	{attribute 'TcIecLibraryType'}
	{attribute 'external_name' := 'F_VN_GetPerspectiveTransformation_GUID_9BE9794E_D7DA_4639_C989_773406D6F2EE'}
	(* Calculate the perspective transformation between four corresponding point pairs. The points mark the corners of the corresponding rectangles. *)
	FUNCTION F_VN_GetPerspectiveTransformation : HRESULT
	VAR_IN_OUT
		aSrcPoints	:	TcVnArray4_Point2_REAL;	(* Source points *)
		aDestPoints	:	TcVnArray4_Point2_REAL;	(* Destination points *)
		aTransformationMatrix	:	TcVnMatrix3x3_LREAL;	(* Resulting transformation matrix *)
	END_VAR
	VAR_INPUT
		hrPrev	:	HRESULT;	(* HRESULT indicating the result of previous operations (If SUCCEEDED(hrPrev) equals false, no operation is executed.) *)
	END_VAR

END_FUNCTION

// Functions/Geometric and Coordinate Transformations/F_VN_Homography

	{attribute 'TcIecLibraryType'}
	{attribute 'external_name' := 'F_VN_Homography_GUID_E5291A1A_EEBB_4859_F9E7_C15E795ADB21'}
	(* Find the homography (perspective transformation) between two planar point sets using RANSAC algorithm. *)
	FUNCTION F_VN_Homography : HRESULT
	VAR_INPUT
		ipSrcPoints	:	ITcVnContainer;	(* Container with at least 4 source points (ContainerType_Vector_TcVnPoint2_REAL) *)
		ipDestPoints	:	ITcVnContainer;	(* Container with destination points (same number as ipSrcPoints, ContainerType_Vector_TcVnPoint2_REAL) *)
	END_VAR
	VAR_IN_OUT
		aPerspectiveTransform	:	TcVnMatrix3x3_LREAL;	(* Returns the perspective transformation matrix, which transforms the source points to the destination points *)
	END_VAR
	VAR_INPUT
		hrPrev	:	HRESULT;	(* HRESULT indicating the result of previous operations (If SUCCEEDED(hrPrev) equals false, no operation is executed.) *)
	END_VAR

END_FUNCTION

// Functions/Geometric and Coordinate Transformations/F_VN_HomographyExp

	{attribute 'TcIecLibraryType'}
	{attribute 'external_name' := 'F_VN_HomographyExp_GUID_CA9C0CB0_39C3_499B_C695_857A7F2AD576'}
	(* Find the homography (perspective transformation) between two planar point sets. (expert function) *)
	FUNCTION F_VN_HomographyExp : HRESULT
	VAR_INPUT
		ipSrcPoints	:	ITcVnContainer;	(* Container with at least 4 source points (ContainerType_Vector_TcVnPoint2_REAL) *)
		ipDestPoints	:	ITcVnContainer;	(* Container with destination points (same number as ipSrcPoints, ContainerType_Vector_TcVnPoint2_REAL) *)
	END_VAR
	VAR_IN_OUT
		aPerspectiveTransform	:	TcVnMatrix3x3_LREAL;	(* Returns the perspective transformation matrix, which transforms the source points to the destination points *)
	END_VAR
	VAR_INPUT
		eAlgorithm	:	ETcVnEstimationAlgorithm;	(* Estimation algorithm *)
		fReprojThreshold	:	LREAL;	(* Maximum allowed reprojection error to treat a point pair as an inlier (only for RANSAC, RHO) *)
		ipInlierMask	:	REFERENCE TO ITcVnContainer;	(* Returns a mask marking the inliers (optional, set to 0 if not required; ContainerType_Vector_SINT; only for RANSAC, LMEDS) *)
		nMaxIterations	:	UDINT;	(* Maximum number of RANSAC iterations *)
		fConfidence	:	LREAL;	(* Confidence (0..1) *)
		hrPrev	:	HRESULT;	(* HRESULT indicating the result of previous operations (If SUCCEEDED(hrPrev) equals false, no operation is executed.) *)
	END_VAR

END_FUNCTION

// Functions/Geometric and Coordinate Transformations/F_VN_InvertAffineTransformation

	{attribute 'TcIecLibraryType'}
	{attribute 'external_name' := 'F_VN_InvertAffineTransformation_GUID_C334F815_EF33_4023_C9C1_C2FEB1CAF8F9'}
	(* Invert a 2D affine transformation matrix. The inverted transformation compensates the affine transformation on an image if it is used in the F_VN_WarpAffine function. *)
	FUNCTION F_VN_InvertAffineTransformation : HRESULT
	VAR_IN_OUT
		aTransformationMatrix	:	TcVnMatrix2x3_LREAL;	(* Source affine transformation matrix *)
		aInvertedTransformationMatrix	:	TcVnMatrix2x3_LREAL;	(* Resulting inverted affine transformation matrix *)
	END_VAR
	VAR_INPUT
		hrPrev	:	HRESULT;	(* HRESULT indicating the result of previous operations (If SUCCEEDED(hrPrev) equals false, no operation is executed.) *)
	END_VAR

END_FUNCTION

// Functions/Geometric and Coordinate Transformations/F_VN_WarpAffine

	{attribute 'TcIecLibraryType'}
	{attribute 'external_name' := 'F_VN_WarpAffine_GUID_78E1DA68_0848_4442_E97A_23AF60C67DC9'}
	(* Apply an affine transformation to an image. *)
	FUNCTION F_VN_WarpAffine : HRESULT
	VAR_INPUT
		ipSrcImage	:	ITcVnImage;	(* Source image *)
		ipDestImage	:	REFERENCE TO ITcVnImage;	(* Destination image (An appropriate image will be created if required.) *)
	END_VAR
	VAR_IN_OUT
		aTransformationMatrix	:	TcVnMatrix2x3_LREAL;	(* Affine transformation matrix *)
	END_VAR
	VAR_INPUT
		hrPrev	:	HRESULT;	(* HRESULT indicating the result of previous operations (If SUCCEEDED(hrPrev) equals false, no operation is executed.) *)
	END_VAR

END_FUNCTION

// Functions/Geometric and Coordinate Transformations/F_VN_PerspectiveTransformation

	{attribute 'TcIecLibraryType'}
	{attribute 'external_name' := 'F_VN_PerspectiveTransformation_GUID_FEECE007_7BAC_4816_C55F_29631736D6C5'}
	(* Apply a perspective transformation (rotation + translation, e.g. from extrinsic calibration) to 3D point coordinates. *)
	FUNCTION F_VN_PerspectiveTransformation : HRESULT
	VAR_INPUT
		ipSrcPoints	:	ITcVnContainer;	(* Container with 3D source points (TcVnPoint3_REAL or TcVnPoint3_LREAL) *)
		ipDestPoints	:	REFERENCE TO ITcVnContainer;	(* Returns the transformed points (same type as ipSrcPoints) *)
	END_VAR
	VAR_IN_OUT
		aRotationMatrix	:	TcVnMatrix3x3_LREAL;	(* 3x3 rotation matrix *)
		aTranslationVector	:	TcVnVector3_LREAL;	(* Translation vector *)
	END_VAR
	VAR_INPUT
		hrPrev	:	HRESULT;	(* HRESULT indicating the result of previous operations (If SUCCEEDED(hrPrev) equals false, no operation is executed.) *)
	END_VAR

END_FUNCTION

// Functions/Geometric and Coordinate Transformations/F_VN_PyramidDown

	{attribute 'TcIecLibraryType'}
	{attribute 'external_name' := 'F_VN_PyramidDown_GUID_FB8B02E5_B7F2_4AD9_D83B_083942D35F0A'}
	(* Downsamples an image to half width and height. *)
	FUNCTION F_VN_PyramidDown : HRESULT
	VAR_INPUT
		ipSrcImage	:	ITcVnImage;	(* Source image *)
		ipDestImage	:	REFERENCE TO ITcVnImage;	(* Destination image (An appropriate destination image will be created if required.) *)
		hrPrev	:	HRESULT;	(* HRESULT indicating the result of previous operations (If SUCCEEDED(hrPrev) equals false, no operation is executed.) *)
	END_VAR

END_FUNCTION

// Functions/Geometric and Coordinate Transformations/F_VN_PyramidUp

	{attribute 'TcIecLibraryType'}
	{attribute 'external_name' := 'F_VN_PyramidUp_GUID_9885070C_2F9E_4CBD_C0E2_B8BDF3FAFC70'}
	(* Upsamples an image to double width and height. *)
	FUNCTION F_VN_PyramidUp : HRESULT
	VAR_INPUT
		ipSrcImage	:	ITcVnImage;	(* Source image *)
		ipDestImage	:	REFERENCE TO ITcVnImage;	(* Destination image (An appropriate destination image will be created if required.) *)
		hrPrev	:	HRESULT;	(* HRESULT indicating the result of previous operations (If SUCCEEDED(hrPrev) equals false, no operation is executed.) *)
	END_VAR

END_FUNCTION

// Functions/Geometric and Coordinate Transformations/F_VN_RemapImageToLogPolarSpace

	{attribute 'TcIecLibraryType'}
	{attribute 'external_name' := 'F_VN_RemapImageToLogPolarSpace_GUID_6E99848D_0ACF_4D69_F527_2E3106AFEFD3'}
	(* Remap an image to log-polar space. *)
	FUNCTION F_VN_RemapImageToLogPolarSpace : HRESULT
	VAR_INPUT
		ipSrcImage	:	ITcVnImage;	(* Source image *)
		ipDestImage	:	REFERENCE TO ITcVnImage;	(* Destination image (Must not be the same as ipSrcImage! An appropriate destination image will be created if required.) *)
	END_VAR
	VAR_IN_OUT
		aCenter	:	TcVnPoint2_REAL;	(* Center point for the transformation *)
	END_VAR
	VAR_INPUT
		hrPrev	:	HRESULT;	(* HRESULT indicating the result of previous operations (If SUCCEEDED(hrPrev) equals false, no operation is executed.) *)
	END_VAR

END_FUNCTION

// Functions/Geometric and Coordinate Transformations/F_VN_RemapImageToLogPolarSpaceExp

	{attribute 'TcIecLibraryType'}
	{attribute 'external_name' := 'F_VN_RemapImageToLogPolarSpaceExp_GUID_9BB5F0DA_4683_4F22_C3F2_6DF6CC34EE46'}
	(* Remap an image to log-polar space. (expert function) *)
	FUNCTION F_VN_RemapImageToLogPolarSpaceExp : HRESULT
	VAR_INPUT
		ipSrcImage	:	ITcVnImage;	(* Source image *)
		ipDestImage	:	REFERENCE TO ITcVnImage;	(* Destination image (Must not be the same as ipSrcImage! An appropriate destination image will be created if required.) *)
	END_VAR
	VAR_IN_OUT
		aCenter	:	TcVnPoint2_REAL;	(* Center point for the transformation *)
	END_VAR
	VAR_INPUT
		fScale	:	LREAL;	(* Magnitude scale parameter, i.e. image width / ln(radius) (set to 0 for auto select) *)
		eInterpolationType	:	ETcVnInterpolationType;	(* Interpolation type *)
		hrPrev	:	HRESULT;	(* HRESULT indicating the result of previous operations (If SUCCEEDED(hrPrev) equals false, no operation is executed.) *)
	END_VAR

END_FUNCTION

// Functions/Geometric and Coordinate Transformations/F_VN_RemapImageToLogPolarSpaceExp2

	{attribute 'TcIecLibraryType'}
	{attribute 'external_name' := 'F_VN_RemapImageToLogPolarSpaceExp2_GUID_D347BCEC_E69F_4A83_E12E_F22818680819'}
	(* Remap an image to log-polar space. (expert function) *)
	FUNCTION F_VN_RemapImageToLogPolarSpaceExp2 : HRESULT
	VAR_INPUT
		ipSrcImage	:	ITcVnImage;	(* Source image *)
		ipDestImage	:	REFERENCE TO ITcVnImage;	(* Destination image (Must not be the same as ipSrcImage! An appropriate destination image will be created if required.) *)
	END_VAR
	VAR_IN_OUT
		aCenter	:	TcVnPoint2_REAL;	(* Center point for the transformation *)
	END_VAR
	VAR_INPUT
		fScale	:	LREAL;	(* Magnitude scale parameter, i.e. image width / ln(radius) (set to 0 for auto select) *)
		eInterpolationType	:	ETcVnInterpolationType;	(* Interpolation type *)
		nDestWidth	:	DINT;	(* Destination image width (set to -1 for source image width, 0 to auto scale to transformed radius, > 0 for a user defined width) *)
		nDestHeight	:	DINT;	(* destination image height (set to -1 for source image height, 0 to auto scale to transformed radius * PI, > 0 for a user defined height) *)
		hrPrev	:	HRESULT;	(* HRESULT indicating the result of previous operations (If SUCCEEDED(hrPrev) equals false, no operation is executed.) *)
	END_VAR

END_FUNCTION

// Functions/Geometric and Coordinate Transformations/F_VN_RemapImageToPolarSpace

	{attribute 'TcIecLibraryType'}
	{attribute 'external_name' := 'F_VN_RemapImageToPolarSpace_GUID_DE45FD10_0322_4630_F43A_30A819E434CD'}
	(* Remap an image to polar space. *)
	FUNCTION F_VN_RemapImageToPolarSpace : HRESULT
	VAR_INPUT
		ipSrcImage	:	ITcVnImage;	(* Source image *)
		ipDestImage	:	REFERENCE TO ITcVnImage;	(* Destination image (Must not be the same as ipSrcImage! An appropriate destination image will be created if required.) *)
	END_VAR
	VAR_IN_OUT
		aCenter	:	TcVnPoint2_REAL;	(* Center point for the transformation *)
	END_VAR
	VAR_INPUT
		hrPrev	:	HRESULT;	(* HRESULT indicating the result of previous operations (If SUCCEEDED(hrPrev) equals false, no operation is executed.) *)
	END_VAR

END_FUNCTION

// Functions/Geometric and Coordinate Transformations/F_VN_RemapImageToPolarSpaceExp

	{attribute 'TcIecLibraryType'}
	{attribute 'external_name' := 'F_VN_RemapImageToPolarSpaceExp_GUID_9860E05D_5A15_4F04_E9E1_22F5EF3B73E2'}
	(* Remap an image to polar space. (expert function) *)
	FUNCTION F_VN_RemapImageToPolarSpaceExp : HRESULT
	VAR_INPUT
		ipSrcImage	:	ITcVnImage;	(* Source image *)
		ipDestImage	:	REFERENCE TO ITcVnImage;	(* Destination image (Must not be the same as ipSrcImage! An appropriate destination image will be created if required.) *)
	END_VAR
	VAR_IN_OUT
		aCenter	:	TcVnPoint2_REAL;	(* Center point for the transformation *)
	END_VAR
	VAR_INPUT
		fMaxRadius	:	LREAL;	(* Maximum radius for the transformation (set to 0 for auto select) *)
		eInterpolationType	:	ETcVnInterpolationType;	(* Interpolation type *)
		hrPrev	:	HRESULT;	(* HRESULT indicating the result of previous operations (If SUCCEEDED(hrPrev) equals false, no operation is executed.) *)
	END_VAR

END_FUNCTION

// Functions/Geometric and Coordinate Transformations/F_VN_RemapImageToPolarSpaceExp2

	{attribute 'TcIecLibraryType'}
	{attribute 'external_name' := 'F_VN_RemapImageToPolarSpaceExp2_GUID_630BAAF6_2143_4E62_F9BA_CD5AAB59C67E'}
	(* Remap an image to polar space. (expert function) *)
	FUNCTION F_VN_RemapImageToPolarSpaceExp2 : HRESULT
	VAR_INPUT
		ipSrcImage	:	ITcVnImage;	(* Source image *)
		ipDestImage	:	REFERENCE TO ITcVnImage;	(* Destination image (Must not be the same as ipSrcImage! An appropriate destination image will be created if required.) *)
	END_VAR
	VAR_IN_OUT
		aCenter	:	TcVnPoint2_REAL;	(* Center point for the transformation *)
	END_VAR
	VAR_INPUT
		fMaxRadius	:	LREAL;	(* Maximum radius for the transformation (set to 0 for auto select) *)
		eInterpolationType	:	ETcVnInterpolationType;	(* Interpolation type *)
		nDestWidth	:	DINT;	(* Destination image width (set to -1 for source image width, 0 to auto scale to transformed radius, > 0 for a user defined width) *)
		nDestHeight	:	DINT;	(* destination image height (set to -1 for source image height, 0 to auto scale to transformed radius * PI, > 0 for a user defined height) *)
		hrPrev	:	HRESULT;	(* HRESULT indicating the result of previous operations (If SUCCEEDED(hrPrev) equals false, no operation is executed.) *)
	END_VAR

END_FUNCTION

// Functions/Geometric and Coordinate Transformations/F_VN_ResizeImage

	{attribute 'TcIecLibraryType'}
	{attribute 'external_name' := 'F_VN_ResizeImage_GUID_ED70CE00_559D_43CE_CB1F_72B9FB8B052F'}
	(* Resize an image using a specific interpolation type. *)
	FUNCTION F_VN_ResizeImage : HRESULT
	VAR_INPUT
		ipSrcImage	:	ITcVnImage;	(* Source image *)
		ipDestImage	:	REFERENCE TO ITcVnImage;	(* Destination image (An appropriate image will be created if required.) *)
		nWidth	:	UDINT;	(* New width *)
		nHeight	:	UDINT;	(* New height *)
		eInterpolationType	:	ETcVnInterpolationType;	(* Interpolation type *)
		hrPrev	:	HRESULT;	(* HRESULT indicating the result of previous operations (If SUCCEEDED(hrPrev) equals false, no operation is executed.) *)
	END_VAR

END_FUNCTION

// Functions/Geometric and Coordinate Transformations/F_VN_ResizeImageExp

	{attribute 'TcIecLibraryType'}
	{attribute 'external_name' := 'F_VN_ResizeImageExp_GUID_377703E0_DC16_4250_DD46_18CED214792B'}
	(* Resize an image using a specific interpolation type while maintaining its aspect ratio. (expert function) *)
	FUNCTION F_VN_ResizeImageExp : HRESULT
	VAR_INPUT
		ipSrcImage	:	ITcVnImage;	(* Source image *)
		ipDestImage	:	REFERENCE TO ITcVnImage;	(* Destination image (An appropriate image will be created if required.) *)
		nWidth	:	UDINT;	(* New width *)
		nHeight	:	UDINT;	(* New height *)
		eInterpolationType	:	ETcVnInterpolationType;	(* Interpolation type *)
		ePaddingMode	:	ETcVnPaddingMode;	(* Image padding mode *)
	END_VAR
	VAR_IN_OUT
		aBorderValue	:	TcVnVector4_LREAL;	(* Border value, if TCVN_PM_LETTERBOX is used *)
	END_VAR
	VAR_INPUT
		hrPrev	:	HRESULT;	(* HRESULT indicating the result of previous operations (If SUCCEEDED(hrPrev) equals false, no operation is executed.) *)
	END_VAR

END_FUNCTION

// Functions/Geometric and Coordinate Transformations/F_VN_RotateImage

	{attribute 'TcIecLibraryType'}
	{attribute 'external_name' := 'F_VN_RotateImage_GUID_8CAB3FB7_5E87_43EF_E423_2C00B8AA20D2'}
	(* Rotate an image by 90, 180, or 270 degrees in clockwise direction. *)
	FUNCTION F_VN_RotateImage : HRESULT
	VAR_INPUT
		ipSrcImage	:	ITcVnImage;	(* Source image *)
		ipDestImage	:	REFERENCE TO ITcVnImage;	(* Destination image (An appropriate image will be created if required.) *)
		eAngle	:	ETcVnRotationAngle;	(* Rotation angle *)
		hrPrev	:	HRESULT;	(* HRESULT indicating the result of previous operations (If SUCCEEDED(hrPrev) equals false, no operation is executed.) *)
	END_VAR

END_FUNCTION

// Functions/Geometric and Coordinate Transformations/F_VN_RotateImageExp

	{attribute 'TcIecLibraryType'}
	{attribute 'external_name' := 'F_VN_RotateImageExp_GUID_A2207F24_DE10_44CD_DD61_03B9D4F8B389'}
	(* Rotate an image by an individual rotation angle in degrees. *)
	FUNCTION F_VN_RotateImageExp : HRESULT
	VAR_INPUT
		ipSrcImage	:	ITcVnImage;	(* Source image *)
		ipDestImage	:	REFERENCE TO ITcVnImage;	(* Destination image (An appropriate image will be created if required.) *)
		fAngleDeg	:	LREAL;	(* Rotation angle in degree (positive: counter-clockwise, negative: clockwise) *)
		bAdjustDestSize	:	BOOL;	(* If true, ipDestImage size is adjusted so that the whole rotated ipSrcImage is contained. Otherwise, ipDestImage size is set to ipSrcImage size. *)
		hrPrev	:	HRESULT;	(* HRESULT indicating the result of previous operations (If SUCCEEDED(hrPrev) equals false, no operation is executed.) *)
	END_VAR

END_FUNCTION

// Functions/Geometric and Coordinate Transformations/F_VN_RotateImageExp2

	{attribute 'TcIecLibraryType'}
	{attribute 'external_name' := 'F_VN_RotateImageExp2_GUID_85F7CE2B_7D57_4E8E_D6F0_120EAB5D6A53'}
	(* Rotate an image by an individual rotation angle in degrees. (expert function) *)
	FUNCTION F_VN_RotateImageExp2 : HRESULT
	VAR_INPUT
		ipSrcImage	:	ITcVnImage;	(* Source image *)
		ipDestImage	:	REFERENCE TO ITcVnImage;	(* Destination image (An appropriate image will be created if required.) *)
		fAngleDeg	:	LREAL;	(* Rotation angle in degree (positive: counter-clockwise, negative: clockwise) *)
		bAdjustDestSize	:	BOOL;	(* If true, ipDestImage size is adjusted so that the whole rotated ipSrcImage is contained. Otherwise, ipDestImage size is set to ipSrcImage size. *)
		eInterpolationType	:	ETcVnInterpolationType;	(* Interpolation method *)
		eBorderInterpolation	:	ETcVnBorderInterpolationMethod;	(* Border interpolation method (ISOLATED not supported) *)
	END_VAR
	VAR_IN_OUT
		aBorderValue	:	TcVnVector4_LREAL;	(* Border value, if CONSTANT is used *)
	END_VAR
	VAR_INPUT
		hrPrev	:	HRESULT;	(* HRESULT indicating the result of previous operations (If SUCCEEDED(hrPrev) equals false, no operation is executed.) *)
	END_VAR

END_FUNCTION

// Functions/Geometric and Coordinate Transformations/F_VN_WarpAffineExp

	{attribute 'TcIecLibraryType'}
	{attribute 'external_name' := 'F_VN_WarpAffineExp_GUID_E5CBC38D_CE6D_4892_FDDC_E6736DBE061C'}
	(* Apply an affine transformation to an image. (expert function) *)
	FUNCTION F_VN_WarpAffineExp : HRESULT
	VAR_INPUT
		ipSrcImage	:	ITcVnImage;	(* Source image *)
		ipDestImage	:	REFERENCE TO ITcVnImage;	(* Destination image (An appropriate image will be created if required.) *)
	END_VAR
	VAR_IN_OUT
		aTransformationMatrix	:	TcVnMatrix2x3_LREAL;	(* Affine transformation matrix *)
	END_VAR
	VAR_INPUT
		nDestWidth	:	UDINT;	(* Width of the destination image *)
		nDestHeight	:	UDINT;	(* Height of the destination image *)
		eInterpolationType	:	ETcVnInterpolationType;	(* Interpolation method *)
		bWarpInverse	:	BOOL;	(* Handle aTransformationMatrix as the inverse transformation *)
		eBorderInterpolation	:	ETcVnBorderInterpolationMethod;	(* Border interpolation method (ISOLATED not supported) *)
		fBorderValue	:	LREAL;	(* Border value, if CONSTANT is used *)
		hrPrev	:	HRESULT;	(* HRESULT indicating the result of previous operations (If SUCCEEDED(hrPrev) equals false, no operation is executed.) *)
	END_VAR

END_FUNCTION

// Functions/Geometric and Coordinate Transformations/F_VN_WarpAffine_Container

	{attribute 'TcIecLibraryType'}
	{attribute 'external_name' := 'F_VN_WarpAffine_Container_GUID_BDA2D4B3_B51A_4A2F_C820_697FB0178013'}
	(* Apply an affine transformation to a container of 2D points. *)
	FUNCTION F_VN_WarpAffine_Container : HRESULT
	VAR_INPUT
		ipSrcPoints	:	ITcVnContainer;	(* Source points (ContainerType_Vector_TcVnPoint2_DINT or ContainerType_Vector_TcVnPoint2_REAL or ContainerType_Vector_TcVnPoint2_LREAL) *)
		ipDestPoints	:	REFERENCE TO ITcVnContainer;	(* Returns the transformed points (same type ID as ipSrcPoints; Non-zero interface pointers are reused.) *)
	END_VAR
	VAR_IN_OUT
		aTransformationMatrix	:	TcVnMatrix2x3_LREAL;	(* Affine transformation matrix *)
	END_VAR
	VAR_INPUT
		hrPrev	:	HRESULT;	(* HRESULT indicating the result of previous operations (If SUCCEEDED(hrPrev) equals false, no operation is executed.) *)
	END_VAR

END_FUNCTION

// Functions/Geometric and Coordinate Transformations/F_VN_WarpAffine_Point

	{attribute 'TcIecLibraryType'}
	{attribute 'external_name' := 'F_VN_WarpAffine_Point_GUID_0C65AB93_8901_4F57_F455_A874377D5041'}
	(* Apply an affine transformation to a 2D point. *)
	FUNCTION F_VN_WarpAffine_Point : HRESULT
	VAR_IN_OUT
		aSrcPoint	:	TcVnPoint2_LREAL;	(* Source point *)
		aDestPoint	:	TcVnPoint2_LREAL;	(* Destination point *)
		aTransformationMatrix	:	TcVnMatrix2x3_LREAL;	(* Affine transformation matrix *)
	END_VAR
	VAR_INPUT
		hrPrev	:	HRESULT;	(* HRESULT indicating the result of previous operations (If SUCCEEDED(hrPrev) equals false, no operation is executed.) *)
	END_VAR

END_FUNCTION

// Functions/Geometric and Coordinate Transformations/F_VN_WarpAffine_Rectangle

	{attribute 'TcIecLibraryType'}
	{attribute 'external_name' := 'F_VN_WarpAffine_Rectangle_GUID_5C0D29CF_C44A_4C24_F34A_859F4FD8ADB8'}
	(* Use an affine transform to warp a rectangle. *)
	FUNCTION F_VN_WarpAffine_Rectangle : HRESULT
	VAR_INPUT
		nTopLeftX	:	UDINT;	(* x coordinate of the top left corner *)
		nTopLeftY	:	UDINT;	(* y coordinate of the top left corner *)
		nBottomRightX	:	UDINT;	(* x coordinate of the bottom right corner *)
		nBottomRightY	:	UDINT;	(* y coordinate of the bottom right corner *)
		ipDestPoints	:	REFERENCE TO ITcVnContainer;	(* Returns the 4 transformed points (ContainerType_Vector_TcVnPoint2_REAL) *)
	END_VAR
	VAR_IN_OUT
		aTransformationMatrix	:	TcVnMatrix2x3_LREAL;	(* Affine transformation matrix *)
	END_VAR
	VAR_INPUT
		hrPrev	:	HRESULT;	(* HRESULT indicating the result of previous operations (If SUCCEEDED(hrPrev) equals false, no operation is executed.) *)
	END_VAR

END_FUNCTION

// Functions/Geometric and Coordinate Transformations/F_VN_WarpPerspective

	{attribute 'TcIecLibraryType'}
	{attribute 'external_name' := 'F_VN_WarpPerspective_GUID_FA579732_BEC2_4958_E42E_5F92911D7AE0'}
	(* Apply a perspective transformation to an image. *)
	FUNCTION F_VN_WarpPerspective : HRESULT
	VAR_INPUT
		ipSrcImage	:	ITcVnImage;	(* Source image *)
		ipDestImage	:	REFERENCE TO ITcVnImage;	(* Destination image (An appropriate image will be created if required.) *)
	END_VAR
	VAR_IN_OUT
		aTransformationMatrix	:	TcVnMatrix3x3_LREAL;	(* Perspective transformation matrix *)
	END_VAR
	VAR_INPUT
		hrPrev	:	HRESULT;	(* HRESULT indicating the result of previous operations (If SUCCEEDED(hrPrev) equals false, no operation is executed.) *)
	END_VAR

END_FUNCTION

// Functions/Geometric and Coordinate Transformations/F_VN_WarpPerspective_Container

	{attribute 'TcIecLibraryType'}
	{attribute 'external_name' := 'F_VN_WarpPerspective_Container_GUID_F182FCB6_9954_46A8_C212_0E4575B35202'}
	(* Apply a perspective transformation to a container of 2D points. *)
	FUNCTION F_VN_WarpPerspective_Container : HRESULT
	VAR_INPUT
		ipSrcPoints	:	ITcVnContainer;	(* Source points (ContainerType_Vector_TcVnPoint2_DINT or ContainerType_Vector_TcVnPoint2_REAL or ContainerType_Vector_TcVnPoint2_LREAL) *)
		ipDestPoints	:	REFERENCE TO ITcVnContainer;	(* Returns the transformed points (same type ID as ipSrcPoints; Non-zero interface pointers are reused.) *)
	END_VAR
	VAR_IN_OUT
		aTransformationMatrix	:	TcVnMatrix3x3_LREAL;	(* Perspective transformation matrix *)
	END_VAR
	VAR_INPUT
		hrPrev	:	HRESULT;	(* HRESULT indicating the result of previous operations (If SUCCEEDED(hrPrev) equals false, no operation is executed.) *)
	END_VAR

END_FUNCTION

// Functions/Geometric and Coordinate Transformations/F_VN_WarpPerspectiveExp

	{attribute 'TcIecLibraryType'}
	{attribute 'external_name' := 'F_VN_WarpPerspectiveExp_GUID_0101B598_6EE4_4C4D_F167_907DFB52670E'}
	(* Apply a perspective transformation to an image. (expert function) *)
	FUNCTION F_VN_WarpPerspectiveExp : HRESULT
	VAR_INPUT
		ipSrcImage	:	ITcVnImage;	(* Source image *)
		ipDestImage	:	REFERENCE TO ITcVnImage;	(* Destination image (An appropriate image will be created if required.) *)
	END_VAR
	VAR_IN_OUT
		aTransformationMatrix	:	TcVnMatrix3x3_LREAL;	(* Perspective transformation matrix *)
	END_VAR
	VAR_INPUT
		nDestWidth	:	UDINT;	(* Width of the destination image *)
		nDestHeight	:	UDINT;	(* Height of the destination image *)
		eInterpolationType	:	ETcVnInterpolationType;	(* Interpolation method *)
		bWarpInverse	:	BOOL;	(* Handle aTransformationMatrix as the inverse transformation *)
		eBorderInterpolation	:	ETcVnBorderInterpolationMethod;	(* Border interpolation method (ISOLATED not supported) *)
		fBorderValue	:	LREAL;	(* Border value, if CONSTANT is used *)
		hrPrev	:	HRESULT;	(* HRESULT indicating the result of previous operations (If SUCCEEDED(hrPrev) equals false, no operation is executed.) *)
	END_VAR

END_FUNCTION

// Functions/Geometric and Coordinate Transformations/F_VN_WarpPerspective_Point

	{attribute 'TcIecLibraryType'}
	{attribute 'external_name' := 'F_VN_WarpPerspective_Point_GUID_0ADF8ADE_46B9_4EEE_EE54_6AF0F99DCBC8'}
	(* Apply a perspective transformation to a 2D point. *)
	FUNCTION F_VN_WarpPerspective_Point : HRESULT
	VAR_IN_OUT
		aSrcPoint	:	TcVnPoint2_LREAL;	(* Source point *)
		aDestPoint	:	TcVnPoint2_LREAL;	(* Destination point *)
		aTransformationMatrix	:	TcVnMatrix3x3_LREAL;	(* Perspective transformation matrix *)
	END_VAR
	VAR_INPUT
		hrPrev	:	HRESULT;	(* HRESULT indicating the result of previous operations (If SUCCEEDED(hrPrev) equals false, no operation is executed.) *)
	END_VAR

END_FUNCTION

// Functions/Geometric and Coordinate Transformations/F_VN_WarpPerspective_Rectangle

	{attribute 'TcIecLibraryType'}
	{attribute 'external_name' := 'F_VN_WarpPerspective_Rectangle_GUID_FCB2B455_A681_4AD4_F5F7_27725716AA61'}
	(* Use a perspective transform to warp a rectangle. *)
	FUNCTION F_VN_WarpPerspective_Rectangle : HRESULT
	VAR_INPUT
		nTopLeftX	:	UDINT;	(* x coordinate of the top left corner *)
		nTopLeftY	:	UDINT;	(* y coordinate of the top left corner *)
		nBottomRightX	:	UDINT;	(* x coordinate of the bottom right corner *)
		nBottomRightY	:	UDINT;	(* y coordinate of the bottom right corner *)
		ipDestPoints	:	REFERENCE TO ITcVnContainer;	(* Returns the 4 transformed points (ContainerType_Vector_TcVnPoint2_REAL) *)
	END_VAR
	VAR_IN_OUT
		aTransformationMatrix	:	TcVnMatrix3x3_LREAL;	(* Perspective transformation matrix *)
	END_VAR
	VAR_INPUT
		hrPrev	:	HRESULT;	(* HRESULT indicating the result of previous operations (If SUCCEEDED(hrPrev) equals false, no operation is executed.) *)
	END_VAR

END_FUNCTION

// Functions/Image Color and Contrast Processing/F_VN_ApplyColorMap

	{attribute 'TcIecLibraryType'}
	{attribute 'external_name' := 'F_VN_ApplyColorMap_GUID_6A737126_4D72_4BCB_EC05_C06460642509'}
	(* Apply a color map to a gray-level image. *)
	FUNCTION F_VN_ApplyColorMap : HRESULT
	VAR_INPUT
		ipSrcImage	:	ITcVnImage;	(* Source image (TCVN_ET_USINT or TCVN_ET_UINT, 1 channel) *)
		ipDestImage	:	REFERENCE TO ITcVnImage;	(* Returns the colored image (TCVN_ET_USINT, 3 channel. An appropriate image will be created if required.) *)
		ipColorMap	:	ITcVnContainer;	(* Color map to be applied to ipSrcImage (ContainerType_Vector_TcVnVector3_REAL with 256 or 65536 elements, dependent on ipSrcImage type). Can be either custom or created with F_VN_GenerateColorMap. *)
		hrPrev	:	HRESULT;	(* HRESULT indicating the result of previous operations (If SUCCEEDED(hrPrev) equals false, no operation is executed.) *)
	END_VAR

END_FUNCTION

// Functions/Image Color and Contrast Processing/F_VN_GenerateColorMap

	{attribute 'TcIecLibraryType'}
	{attribute 'external_name' := 'F_VN_GenerateColorMap_GUID_74A0CE66_74B2_42A4_C756_B0F27E943F8E'}
	(* Generates a pre-defined color map. *)
	FUNCTION F_VN_GenerateColorMap : HRESULT
	VAR_INPUT
		ipColorMap	:	REFERENCE TO ITcVnContainer;	(* Returns the color map (ContainerType_Vector_TcVnVector3_REAL with 256 or 65536 elements) *)
		eColorMap	:	ETcVnColorMap;	(* Selects a color map (similar to GNU Octave/MATLAB types) *)
		eColorMapSize	:	ETcVnColorMapSize;	(* Defines how many elements the generated color map should have *)
		hrPrev	:	HRESULT;	(* HRESULT indicating the result of previous operations (If SUCCEEDED(hrPrev) equals false, no operation is executed.) *)
	END_VAR

END_FUNCTION

// Functions/Image Color and Contrast Processing/F_VN_ApplyLut

	{attribute 'TcIecLibraryType'}
	{attribute 'external_name' := 'F_VN_ApplyLut_GUID_68C1FC50_DE6A_4FE0_E3D5_AD24FA9B5417'}
	(* Apply a lookup table to an image to manipulate its colors. *)
	FUNCTION F_VN_ApplyLut : HRESULT
	VAR_INPUT
		ipSrcImage	:	ITcVnImage;	(* Source image (1-4 channels of 8 or 16 bit types SINT, USINT, INT, UINT) *)
		ipDestImage	:	REFERENCE TO ITcVnImage;	(* Returns the result image (same size, type and channels as ipSrcImage. An appropriate image will be created if required.) *)
		ipLut	:	ITcVnContainer;	(* Lookup table with elements matching ipSrcImage type and either 256 (8 bit images) or 65536 (16 bit images) elements. E.g. ContainerType_Vector_USINT for 1-4 channel USINT image (in this case, the same lookup values are used for each channel) or ContainerType_Vector_TcVnVector3_USINT for a 3 channel USINT image (in this case, each channel uses an individual lookup value).
						 *)
		hrPrev	:	HRESULT;	(* HRESULT indicating the result of previous operations (If SUCCEEDED(hrPrev) equals false, no operation is executed.) *)
	END_VAR

END_FUNCTION

// Functions/Image Color and Contrast Processing/F_VN_Clahe

	{attribute 'TcIecLibraryType'}
	{attribute 'external_name' := 'F_VN_Clahe_GUID_5A201C60_0417_4646_D4DD_B850B6060DD9'}
	(* Apply Constrast Limited Adaptive Histogram Equalization. This applies local histogram equalization to individual tiles. *)
	FUNCTION F_VN_Clahe : HRESULT
	VAR_INPUT
		ipSrcImage	:	ITcVnImage;	(* Source image (TCVN_ET_USINT or TCVN_ET_UINT, 1 channel) *)
		ipDestImage	:	REFERENCE TO ITcVnImage;	(* Returns the resulting image (An appropriate image will be created if required.) *)
		hrPrev	:	HRESULT;	(* HRESULT indicating the result of previous operations (If SUCCEEDED(hrPrev) equals false, no operation is executed.) *)
	END_VAR

END_FUNCTION

// Functions/Image Color and Contrast Processing/F_VN_ClaheExp

	{attribute 'TcIecLibraryType'}
	{attribute 'external_name' := 'F_VN_ClaheExp_GUID_E01C29C2_6F3D_4620_E8A1_F87756DA5EF7'}
	(* Apply Constrast Limited Adaptive Histogram Equalization. This applies local histogram equalization to individual tiles. (expert function) *)
	FUNCTION F_VN_ClaheExp : HRESULT
	VAR_INPUT
		ipSrcImage	:	ITcVnImage;	(* Source image (TCVN_ET_USINT or TCVN_ET_UINT, 1 channel) *)
		ipDestImage	:	REFERENCE TO ITcVnImage;	(* Returns the resulting image (An appropriate image will be created if required.) *)
		fClipLimit	:	LREAL;	(* Threshold for contrast limit (set to <= 0 to disable clipping) *)
		nTilesX	:	UDINT;	(* Number of tiles in x direction *)
		nTilesY	:	UDINT;	(* Number of tiles in y direction *)
		hrPrev	:	HRESULT;	(* HRESULT indicating the result of previous operations (If SUCCEEDED(hrPrev) equals false, no operation is executed.) *)
	END_VAR

END_FUNCTION

// Functions/Image Color and Contrast Processing/F_VN_ConvertColorSpace

	{attribute 'TcIecLibraryType'}
	{attribute 'external_name' := 'F_VN_ConvertColorSpace_GUID_0C9A6943_44C8_4F3F_E050_0540D257B30D'}
	(* Convert image from one color space to another. *)
	FUNCTION F_VN_ConvertColorSpace : HRESULT
	VAR_INPUT
		ipSrcImage	:	ITcVnImage;	(* Source image *)
		ipDestImage	:	REFERENCE TO ITcVnImage;	(* Destination image (An appropriate destination image will be created if required.) *)
		eTransform	:	ETcVnColorSpaceTransform;	(* Transforms to be applied *)
		hrPrev	:	HRESULT;	(* HRESULT indicating the result of previous operations (If SUCCEEDED(hrPrev) equals false, no operation is executed.) *)
	END_VAR

END_FUNCTION

// Functions/Image Color and Contrast Processing/F_VN_GenerateCustomColorMap

	{attribute 'TcIecLibraryType'}
	{attribute 'external_name' := 'F_VN_GenerateCustomColorMap_GUID_1094D0C8_CFDF_428E_D6CA_794FDFCF1A89'}
	(* Generate a custom color map by interpolating between user defined colors (equally distributed, linear for each channel). *)
	FUNCTION F_VN_GenerateCustomColorMap : HRESULT
	VAR_INPUT
		ipColorMap	:	REFERENCE TO ITcVnContainer;	(* Returns the color map (ContainerType_Vector_TcVnVector3_REAL with 256 or 65536 elements) *)
		ipInitialColors	:	ITcVnContainer;	(* User defined colors (ContainerType_Vector_TcVnVector3_REAL, at least 2 elements) *)
		eColorMapSize	:	ETcVnColorMapSize;	(* Defines how many elements the generated color map should have *)
		hrPrev	:	HRESULT;	(* HRESULT indicating the result of previous operations (If SUCCEEDED(hrPrev) equals false, no operation is executed.) *)
	END_VAR

END_FUNCTION

// Functions/Image Color and Contrast Processing/F_VN_Histogram

	{attribute 'TcIecLibraryType'}
	{attribute 'external_name' := 'F_VN_Histogram_GUID_7CD52F24_6A0E_4240_F662_690EEE885C29'}
	(* Calculate the (multi-channel) histogram of an image. *)
	FUNCTION F_VN_Histogram : HRESULT
	VAR_INPUT
		ipSrcImage	:	ITcVnImage;	(* Source image *)
		ipDestHistogram	:	REFERENCE TO ITcVnContainer;	(* Returns a container with a multi-channel histogram, where every channel is represented as a vector of UDINT (ContainerType_Vector_Vector_UDINT. Non-zero interface pointers are reused.) *)
		hrPrev	:	HRESULT;	(* HRESULT indicating the result of previous operations (If SUCCEEDED(hrPrev) equals false, no operation is executed.) *)
	END_VAR

END_FUNCTION

// Functions/Image Color and Contrast Processing/F_VN_HistogramExp

	{attribute 'TcIecLibraryType'}
	{attribute 'external_name' := 'F_VN_HistogramExp_GUID_F7FF4E9D_8461_4537_D0B5_042BFE2DC671'}
	(* Calculate the (multi-channel) histogram of an image. (expert function) *)
	FUNCTION F_VN_HistogramExp : HRESULT
	VAR_INPUT
		ipSrcImage	:	ITcVnImage;	(* Source image *)
		ipDestHistogram	:	REFERENCE TO ITcVnContainer;	(* Returns a container with a multi-channel histogram, where every channel is represented as a vector of UDINT (ContainerType_Vector_Vector_UDINT. Non-zero interface pointers are reused.) *)
	END_VAR
	VAR_IN_OUT
		nBins	:	UDINT;	(* Desired number of bins or 0 to keep the default for the corresponding image format (in) and default number of bins (out) *)
		fLowerBound	:	LREAL;	(* Lower (inclusive) boundary of the 0-th histogram bin (in), or receive the default if fLowerBound AND fUpperBound are set to 0 (out) *)
		fUpperBound	:	LREAL;	(* Upper (exclusive) boundary of the last histogram bin nBins-1 (in), or receive the default if fLowerBound AND fUpperBound are set to 0 (out) *)
	END_VAR
	VAR_INPUT
		ipMask	:	ITcVnImage;	(* Source image mask (TCVN_ET_USINT, 1 channel. Mask is optional, set to 0 if not required.) *)
		hrPrev	:	HRESULT;	(* HRESULT indicating the result of previous operations (If SUCCEEDED(hrPrev) equals false, no operation is executed.) *)
	END_VAR

END_FUNCTION

// Functions/Image Color and Contrast Processing/F_VN_HistogramEqualization

	{attribute 'TcIecLibraryType'}
	{attribute 'external_name' := 'F_VN_HistogramEqualization_GUID_D1159D57_C8FC_47EA_ED0E_899FCA521D1C'}
	(* Equalize the histogram of a grayscale or rgb image, which normalizes the brightness and improves the contrast. *)
	FUNCTION F_VN_HistogramEqualization : HRESULT
	VAR_INPUT
		ipSrcImage	:	ITcVnImage;	(* Source image (USINT) *)
		ipDestImage	:	REFERENCE TO ITcVnImage;	(* Destination image (An appropriate destination image will be created if required.) *)
		hrPrev	:	HRESULT;	(* HRESULT indicating the result of previous operations (If SUCCEEDED(hrPrev) equals false, no operation is executed.) *)
	END_VAR

END_FUNCTION

// Functions/Image Color and Contrast Processing/F_VN_HistogramEqualizationExp

	{attribute 'TcIecLibraryType'}
	{attribute 'external_name' := 'F_VN_HistogramEqualizationExp_GUID_BB06441D_3237_48E2_C065_F679AD24D02A'}
	(* Equalize the histogram of a grayscale or color image, which normalizes the brightness and improves the contrast. (expert function) 
	The channel index that should be equalized has to be specified (-1 expects a RGB image, converts it to YCbCr, equalizes the Y channel and converts the image back to RGB).  *)
	FUNCTION F_VN_HistogramEqualizationExp : HRESULT
	VAR_INPUT
		ipSrcImage	:	ITcVnImage;	(* Source image (USINT) *)
		ipDestImage	:	REFERENCE TO ITcVnImage;	(* Destination image (An appropriate destination image will be created if required.) *)
		nChannelIdx	:	INT;	(* Index of the image channel that should be equalized (-1 expects a RGB image, converts it to YCbCr, equalizes the Y channel and converts the image back to RGB) *)
		hrPrev	:	HRESULT;	(* HRESULT indicating the result of previous operations (If SUCCEEDED(hrPrev) equals false, no operation is executed.) *)
	END_VAR

END_FUNCTION

// Functions/Image Color and Contrast Processing/F_VN_InvertImageColor

	{attribute 'TcIecLibraryType'}
	{attribute 'external_name' := 'F_VN_InvertImageColor_GUID_020EB12F_578C_482E_E344_884020060F01'}
	(* Invert the color of an image.
          For signed integer or negative floating point values, only the signs will be switched.
          If the image contains only positive floating point values, each pixel value is subtracted from the maximum available pixel value (or 1.0, whatever is higher). *)
	FUNCTION F_VN_InvertImageColor : HRESULT
	VAR_INPUT
		ipSrcImage	:	ITcVnImage;	(* Source image *)
		ipDestImage	:	REFERENCE TO ITcVnImage;	(* Destination image (An appropriate image will be created if required.) *)
		hrPrev	:	HRESULT;	(* HRESULT indicating the result of previous operations (If SUCCEEDED(hrPrev) equals false, no operation is executed.) *)
	END_VAR

END_FUNCTION

// Functions/Image Color and Contrast Processing/F_VN_InvertImageColorExp

	{attribute 'TcIecLibraryType'}
	{attribute 'external_name' := 'F_VN_InvertImageColorExp_GUID_ED78A235_36B4_4884_D00B_D4AF8582CECD'}
	(* Invert the color of an image. (expert function)
          For signed integer or negative floating point values, only the signs will be switched.
          If the image contains only positive floating point values, each pixel value is subtracted from the maximum available pixel value (or 1.0, whatever is higher). *)
	FUNCTION F_VN_InvertImageColorExp : HRESULT
	VAR_INPUT
		ipSrcImage	:	ITcVnImage;	(* Source image *)
		ipDestImage	:	REFERENCE TO ITcVnImage;	(* Destination image (An appropriate image will be created if required.) *)
		fMaxValue	:	LREAL;	(* Maximum pixel value (e.g. if a 16 bit image contains 12 bit values). -1 means the default values are used. *)
		hrPrev	:	HRESULT;	(* HRESULT indicating the result of previous operations (If SUCCEEDED(hrPrev) equals false, no operation is executed.) *)
	END_VAR

END_FUNCTION

// Functions/Image Color and Contrast Processing/F_VN_NormalizeImage

	{attribute 'TcIecLibraryType'}
	{attribute 'external_name' := 'F_VN_NormalizeImage_GUID_347BC85A_B624_4984_D90F_B69C35030699'}
	(* Normalize an image regarding its value range (e.g. stretch pixel values [50..150] to full range [0..255]). *)
	FUNCTION F_VN_NormalizeImage : HRESULT
	VAR_INPUT
		ipSrcImage	:	ITcVnImage;	(* Source image *)
		ipDestImage	:	REFERENCE TO ITcVnImage;	(* Destination image (An appropriate destination image will be created if required.) *)
		hrPrev	:	HRESULT;	(* HRESULT indicating the result of previous operations (If SUCCEEDED(hrPrev) equals false, no operation is executed.) *)
	END_VAR

END_FUNCTION

// Functions/Image Color and Contrast Processing/F_VN_NormalizeImageExp

	{attribute 'TcIecLibraryType'}
	{attribute 'external_name' := 'F_VN_NormalizeImageExp_GUID_CC978FB6_F368_4C0E_FC1E_10915138DCD5'}
	(* Normalize an image regarding its value range (e.g. stretch pixel values [50..150] to full range [0..255]) or scale the values regarding a specific normalization (e.g. L2-norm). (expert function) *)
	FUNCTION F_VN_NormalizeImageExp : HRESULT
	VAR_INPUT
		ipSrcImage	:	ITcVnImage;	(* Source image *)
		ipDestImage	:	REFERENCE TO ITcVnImage;	(* Destination image (An appropriate destination image will be created if required.) *)
		fAlpha	:	LREAL;	(* Lower range boundary (in case of normalizing the value range) or value to normalize to (||ipDestImage|| = fAlpha) *)
		fBeta	:	LREAL;	(* Upper range boundary (in case of normalizing the value range) *)
		eNormType	:	ETcVnNormalizationType;	(* Normalization type (only INF, L1, L2 or MINMAX) *)
		eDestType	:	ETcVnElementType;	(* Destination image depth (usually SAME_AS_SOURCE) *)
		ipMask	:	ITcVnImage;	(* Mask to restrict the normalization to specific pixel positions (set 0 to normalize the whole image) *)
		hrPrev	:	HRESULT;	(* HRESULT indicating the result of previous operations (If SUCCEEDED(hrPrev) equals false, no operation is executed.) *)
	END_VAR

END_FUNCTION

// Functions/Image Color and Contrast Processing/F_VN_NormalizeImageForDisplay

	{attribute 'TcIecLibraryType'}
	{attribute 'external_name' := 'F_VN_NormalizeImageForDisplay_GUID_6F8B2BD9_79E6_45D9_DEBC_DEE2DCBDF507'}
	(* Normalize an image for display, i.e. scale it to the full value range of the underlying data type (-1 to 1 for floating point). *)
	FUNCTION F_VN_NormalizeImageForDisplay : HRESULT
	VAR_INPUT
		ipSrcImage	:	ITcVnImage;	(* Source image *)
		ipDestImage	:	REFERENCE TO ITcVnImage;	(* Destination image (An appropriate destination image will be created if required.) *)
		eSignedNormalization	:	ETcVnSignedNormalization;	(* Option for normalizing signed values *)
		hrPrev	:	HRESULT;	(* HRESULT indicating the result of previous operations (If SUCCEEDED(hrPrev) equals false, no operation is executed.) *)
	END_VAR

END_FUNCTION

// Functions/Image Color and Contrast Processing/F_VN_ReferenceColorSimilarity_ITcVnColorModel

	{attribute 'TcIecLibraryType'}
	{attribute 'external_name' := 'F_VN_ReferenceColorSimilarity_ITcVnColorModel_GUID_1FADFE82_D14E_4C9E_E66A_E033990D018A'}
	(* Computes the similarity to a reference color model for each pixel in the source image. *)
	FUNCTION F_VN_ReferenceColorSimilarity_ITcVnColorModel : HRESULT
	VAR_INPUT
		ipSrcImage	:	ITcVnImage;	(* RGB source image (USINT, 3 channels) *)
		ipDestImage	:	REFERENCE TO ITcVnImage;	(* Returns the similarity to ipColorModel for each pixel in ipSrcImage (USINT, 1 channel. An appropriate destination image will be created if required.) *)
		ipColorModel	:	ITcVnColorModel;	(* Color model *)
		hrPrev	:	HRESULT;	(* HRESULT indicating the result of previous operations (If SUCCEEDED(hrPrev) equals false, no operation is executed.) *)
	END_VAR

END_FUNCTION

// Interfaces/Machine Learning/ITcVnColorModel

	(* Interface to train and classify an image color. *)
	{attribute 'c++_compatible'}
	{attribute 'vtable_order' := 'TrainImageColor;ClassifyImageColor'}
	INTERFACE ITcVnColorModel EXTENDS ITcVnMlModel


(* Train the color of the provided image. *)
	{attribute 'c++_compatible'}
	{attribute 'minimal_input_size' := '4'}
	{attribute 'pack_mode' := '4'}
	METHOD TrainImageColor : HRESULT
	VAR_INPUT
		ipSrcImage : ITcVnImage;
		nDifferentColors : UDINT;
		ipMask : ITcVnImage;
		nSkipPixels : UDINT;
	END_VAR
END_METHOD


(* Compute the similarity of each image pixel to the trained reference color. *)
	{attribute 'c++_compatible'}
	{attribute 'minimal_input_size' := '4'}
	{attribute 'pack_mode' := '4'}
	METHOD ClassifyImageColor : HRESULT
	VAR_INPUT
		ipSrcImage : ITcVnImage;
		pipDestImage : POINTER TO ITcVnImage;
		fVariance : REAL;
		fLuminanceWeight : REAL;
	END_VAR
END_METHOD

END_INTERFACE

// Functions/Image Color and Contrast Processing/F_VN_ReferenceColorSimilarityExp_ITcVnColorModel

	{attribute 'TcIecLibraryType'}
	{attribute 'external_name' := 'F_VN_ReferenceColorSimilarityExp_ITcVnColorModel_GUID_1BB1CE39_58BF_4D29_CCD3_3E96241740FE'}
	(* Computes the similarity to a reference color model for each pixel in the source image. (expert function) *)
	FUNCTION F_VN_ReferenceColorSimilarityExp_ITcVnColorModel : HRESULT
	VAR_INPUT
		ipSrcImage	:	ITcVnImage;	(* RGB source image (USINT, 3 channels) *)
		ipDestImage	:	REFERENCE TO ITcVnImage;	(* Returns the similarity to ipColorModel for each pixel in ipSrcImage (USINT, 1 channel. An appropriate destination image will be created if required.) *)
		ipColorModel	:	ITcVnColorModel;	(* Color model *)
		fVariance	:	REAL;	(* Allowed color variance (0.1 - 0.3 might be a good start to try) *)
		fLuminanceWeight	:	REAL;	(* Weight the impact of the luminance ([0..1], e.g. set to 0 to be more resistant to unequal illumination, but might be required to differentiate between some colors. Ignored if ipColorModel is of type RGB.) *)
		hrPrev	:	HRESULT;	(* HRESULT indicating the result of previous operations (If SUCCEEDED(hrPrev) equals false, no operation is executed.) *)
	END_VAR

END_FUNCTION

// Functions/Image Color and Contrast Processing/F_VN_ReferenceColorSimilarity_ITcVnMlModel

	{attribute 'TcIecLibraryType'}
	{attribute 'external_name' := 'F_VN_ReferenceColorSimilarity_ITcVnMlModel_GUID_4FC0852C_93D2_43AC_D10C_06008C68329E'}
	(* Computes the similarity to a reference color model for each pixel in the source image. *)
	FUNCTION F_VN_ReferenceColorSimilarity_ITcVnMlModel : HRESULT
	VAR_INPUT
		ipSrcImage	:	ITcVnImage;	(* RGB source image (USINT, 3 channels) *)
		ipDestImage	:	REFERENCE TO ITcVnImage;	(* Returns the similarity to ipColorModel for each pixel in ipSrcImage (USINT, 1 channel. An appropriate destination image will be created if required.) *)
		ipColorModel	:	ITcVnMlModel;	(* Color model *)
		hrPrev	:	HRESULT;	(* HRESULT indicating the result of previous operations (If SUCCEEDED(hrPrev) equals false, no operation is executed.) *)
	END_VAR

END_FUNCTION

// Functions/Image Color and Contrast Processing/F_VN_ReferenceColorSimilarityExp_ITcVnMlModel

	{attribute 'TcIecLibraryType'}
	{attribute 'external_name' := 'F_VN_ReferenceColorSimilarityExp_ITcVnMlModel_GUID_6D1CFD8E_95DC_4639_E165_D4A97C86BCDB'}
	(* Computes the similarity to a reference color model for each pixel in the source image. (expert function) *)
	FUNCTION F_VN_ReferenceColorSimilarityExp_ITcVnMlModel : HRESULT
	VAR_INPUT
		ipSrcImage	:	ITcVnImage;	(* RGB source image (USINT, 3 channels) *)
		ipDestImage	:	REFERENCE TO ITcVnImage;	(* Returns the similarity to ipColorModel for each pixel in ipSrcImage (USINT, 1 channel. An appropriate destination image will be created if required.) *)
		ipColorModel	:	ITcVnMlModel;	(* Color model *)
		fVariance	:	REAL;	(* Allowed color variance (0.1 - 0.3 might be a good start to try) *)
		fLuminanceWeight	:	REAL;	(* Weight the impact of the luminance ([0..1], e.g. set to 0 to be more resistant to unequal illumination, but might be required to differentiate between some colors. Ignored if ipColorModel is of type RGB.) *)
		hrPrev	:	HRESULT;	(* HRESULT indicating the result of previous operations (If SUCCEEDED(hrPrev) equals false, no operation is executed.) *)
	END_VAR

END_FUNCTION

// Functions/Image Color and Contrast Processing/F_VN_ReferenceColorSimilarity_TcVnVector3_LREAL

	{attribute 'TcIecLibraryType'}
	{attribute 'external_name' := 'F_VN_ReferenceColorSimilarity_TcVnVector3_LREAL_GUID_CF4D0FF1_E042_456A_D9AF_1425509594A5'}
	(* Computes the similarity to a reference color for each pixel in the source image. *)
	FUNCTION F_VN_ReferenceColorSimilarity_TcVnVector3_LREAL : HRESULT
	VAR_INPUT
		ipSrcImage	:	ITcVnImage;	(* RGB source image (USINT, 3 channels) *)
		ipDestImage	:	REFERENCE TO ITcVnImage;	(* Returns the similarity to aRefColor for each pixel in ipSrcImage (USINT, 1 channel. An appropriate destination image will be created if required.) *)
	END_VAR
	VAR_IN_OUT
		aRefColor	:	TcVnVector3_LREAL;	(* Reference color (RGB, [0..255]) *)
	END_VAR
	VAR_INPUT
		hrPrev	:	HRESULT;	(* HRESULT indicating the result of previous operations (If SUCCEEDED(hrPrev) equals false, no operation is executed.) *)
	END_VAR

END_FUNCTION

// Functions/Image Color and Contrast Processing/F_VN_ReferenceColorSimilarityExp_TcVnVector3_LREAL

	{attribute 'TcIecLibraryType'}
	{attribute 'external_name' := 'F_VN_ReferenceColorSimilarityExp_TcVnVector3_LREAL_GUID_E6C624F4_C3A4_4FBF_ED77_4736B9F40CB1'}
	(* Computes the similarity to a reference color for each pixel in the source image. (expert function) *)
	FUNCTION F_VN_ReferenceColorSimilarityExp_TcVnVector3_LREAL : HRESULT
	VAR_INPUT
		ipSrcImage	:	ITcVnImage;	(* RGB source image (USINT, 3 channels) *)
		ipDestImage	:	REFERENCE TO ITcVnImage;	(* Returns the similarity to aRefColor for each pixel in ipSrcImage (USINT, 1 channel. An appropriate destination image will be created if required.) *)
	END_VAR
	VAR_IN_OUT
		aRefColor	:	TcVnVector3_LREAL;	(* Reference color (RGB, [0..255]) *)
	END_VAR
	VAR_INPUT
		fVariance	:	REAL;	(* Allowed color variance (0.1 - 0.3 might be a good start to try) *)
		fLuminanceWeight	:	REAL;	(* Weight the impact of the luminance ([0..1], e.g. set to 0 to be more resistant to unequal illumination, but might be required to differentiate between some colors) *)
		hrPrev	:	HRESULT;	(* HRESULT indicating the result of previous operations (If SUCCEEDED(hrPrev) equals false, no operation is executed.) *)
	END_VAR

END_FUNCTION

// Functions/Image Color and Contrast Processing/F_VN_TrainImageColor

	{attribute 'TcIecLibraryType'}
	{attribute 'external_name' := 'F_VN_TrainImageColor_GUID_3734521A_E642_45F7_EDF9_CFC53B23EA15'}
	(* Create a new color model, describing the image color. *)
	FUNCTION F_VN_TrainImageColor : HRESULT
	VAR_INPUT
		ipSrcImage	:	ITcVnImage;	(* Source image (3 channels (RGB) of type USINT) *)
		ipColorModel	:	REFERENCE TO ITcVnColorModel;	(* Returns the color model *)
		nDifferentColors	:	UDINT;	(* Number of different colors to distinguish *)
		hrPrev	:	HRESULT;	(* HRESULT indicating the result of previous operations (If SUCCEEDED(hrPrev) equals false, no operation is executed.) *)
	END_VAR

END_FUNCTION

// Functions/Image Color and Contrast Processing/F_VN_TrainImageColorExp

	{attribute 'TcIecLibraryType'}
	{attribute 'external_name' := 'F_VN_TrainImageColorExp_GUID_54E1D1B3_7DE1_4285_CAE7_9383E286C3EC'}
	(* Create a new color model, describing the image color. (expert function) *)
	FUNCTION F_VN_TrainImageColorExp : HRESULT
	VAR_INPUT
		ipSrcImage	:	ITcVnImage;	(* Source image (3 channels (RGB) of type USINT) *)
		ipColorModel	:	REFERENCE TO ITcVnColorModel;	(* Returns the color model *)
		nDifferentColors	:	UDINT;	(* Number of different colors to distinguish *)
		eMethod	:	ETcVnColorTrainingMethod;	(* Color training method *)
		ipMask	:	ITcVnImage;	(* Optional image mask (1 channel of type USINT, set to 0 if not required) *)
		nSkipPixels	:	UDINT;	(* Number of pixels to skip between each evaluated color sample (to achieve a better performance). 0 takes every pixel into account and tends to be more accurate. *)
		hrPrev	:	HRESULT;	(* HRESULT indicating the result of previous operations (If SUCCEEDED(hrPrev) equals false, no operation is executed.) *)
	END_VAR

END_FUNCTION

// Functions/Image Color and Contrast Processing/F_VN_TrainImageColorExp2

	{attribute 'TcIecLibraryType'}
	{attribute 'external_name' := 'F_VN_TrainImageColorExp2_GUID_31D0944A_7507_4A27_D890_EEC95A07A6BA'}
	(* Create a new color model, describing the image color. (expert function) *)
	FUNCTION F_VN_TrainImageColorExp2 : HRESULT
	VAR_INPUT
		ipSrcImage	:	ITcVnImage;	(* Source image (3 channels (RGB) of type USINT) *)
		ipColorModel	:	REFERENCE TO ITcVnColorModel;	(* Returns the color model *)
		nDifferentColors	:	UDINT;	(* Maximum number of different colors to distinguish (if LBG is used as a clustering algorithm, the result might have less different colors, depending on nMaxClusterRadius) *)
		eMethod	:	ETcVnColorTrainingMethod;	(* Color training method *)
		ipMask	:	ITcVnImage;	(* Optional image mask (1 channel of type USINT, set to 0 if not required) *)
		nSkipPixels	:	UDINT;	(* Number of pixels to skip between each evaluated color sample (to achieve a better performance). 0 takes every pixel into account and tends to be more accurate. *)
		eClusteringAlgorithm	:	ETcVnClusteringAlgorithm;	(* Clustering algorithm *)
		nMaxClusterRadius	:	DINT;	(* Only used for the LBG clustering algorithm. Maximum allowed radius (> 0) of a single cluster, i.e. clusters with a higher radius will be split into smaller ones, until a global number of nDifferentColors is reached. *)
		bSingleSplitSteps	:	BOOL;	(* Only used for the LBG clustering algorithm. If true, the global optimization is always run after a single cluster has been split. If false, several clusters are split within the same step before applying the global optimization. Applying the global optimization less often is faster, but can lead to less optimal results, especially having 2 nearby clusters that could be represented by 1) *)
		hrPrev	:	HRESULT;	(* HRESULT indicating the result of previous operations (If SUCCEEDED(hrPrev) equals false, no operation is executed.) *)
	END_VAR

END_FUNCTION

// Functions/Image Color and Contrast Processing/F_VN_TrainImageColor_ITcVnMlModel

	{attribute 'TcIecLibraryType'}
	{attribute 'external_name' := 'F_VN_TrainImageColor_ITcVnMlModel_GUID_7C37521A_6541_427D_DFD3_8CF85F605412'}
	(* Create a new color model, describing the image color. *)
	FUNCTION F_VN_TrainImageColor_ITcVnMlModel : HRESULT
	VAR_INPUT
		ipSrcImage	:	ITcVnImage;	(* Source image (3 channels (RGB) of type USINT) *)
		ipColorModel	:	REFERENCE TO ITcVnMlModel;	(* Returns the color model *)
		nDifferentColors	:	UDINT;	(* Number of different colors to distinguish *)
		hrPrev	:	HRESULT;	(* HRESULT indicating the result of previous operations (If SUCCEEDED(hrPrev) equals false, no operation is executed.) *)
	END_VAR

END_FUNCTION

// Functions/Image Color and Contrast Processing/F_VN_TrainImageColorExp_ITcVnMlModel

	{attribute 'TcIecLibraryType'}
	{attribute 'external_name' := 'F_VN_TrainImageColorExp_ITcVnMlModel_GUID_DFD92614_2A08_40E9_E0C0_263BFD1F8FEC'}
	(* Create a new color model, describing the image color. (expert function) *)
	FUNCTION F_VN_TrainImageColorExp_ITcVnMlModel : HRESULT
	VAR_INPUT
		ipSrcImage	:	ITcVnImage;	(* Source image (3 channels (RGB) of type USINT) *)
		ipColorModel	:	REFERENCE TO ITcVnMlModel;	(* Returns the color model *)
		nDifferentColors	:	UDINT;	(* Number of different colors to distinguish *)
		eMethod	:	ETcVnColorTrainingMethod;	(* Color training method *)
		ipMask	:	ITcVnImage;	(* Optional image mask (1 channel of type USINT, set to 0 if not required) *)
		nSkipPixels	:	UDINT;	(* Number of pixels to skip between each evaluated color sample (to achieve a better performance). 0 takes every pixel into account and tends to be more accurate. *)
		hrPrev	:	HRESULT;	(* HRESULT indicating the result of previous operations (If SUCCEEDED(hrPrev) equals false, no operation is executed.) *)
	END_VAR

END_FUNCTION

// Functions/Image Color and Contrast Processing/F_VN_TrainImageColorExp2_ITcVnMlModel

	{attribute 'TcIecLibraryType'}
	{attribute 'external_name' := 'F_VN_TrainImageColorExp2_ITcVnMlModel_GUID_67E39DCF_86FC_483C_D31D_175338992E5B'}
	(* Create a new color model, describing the image color. (expert function) *)
	FUNCTION F_VN_TrainImageColorExp2_ITcVnMlModel : HRESULT
	VAR_INPUT
		ipSrcImage	:	ITcVnImage;	(* Source image (3 channels (RGB) of type USINT) *)
		ipColorModel	:	REFERENCE TO ITcVnMlModel;	(* Returns the color model *)
		nDifferentColors	:	UDINT;	(* Maximum number of different colors to distinguish (if LBG is used as a clustering algorithm, the result might have less different colors, depending on nMaxClusterRadius) *)
		eMethod	:	ETcVnColorTrainingMethod;	(* Color training method *)
		ipMask	:	ITcVnImage;	(* Optional image mask (1 channel of type USINT, set to 0 if not required) *)
		nSkipPixels	:	UDINT;	(* Number of pixels to skip between each evaluated color sample (to achieve a better performance). 0 takes every pixel into account and tends to be more accurate. *)
		eClusteringAlgorithm	:	ETcVnClusteringAlgorithm;	(* Clustering algorithm *)
		nMaxClusterRadius	:	DINT;	(* Only used for the LBG clustering algorithm. Maximum allowed radius (> 0) of a single cluster, i.e. clusters with a higher radius will be split into smaller ones, until a global number of nDifferentColors is reached. *)
		bSingleSplitSteps	:	BOOL;	(* Only used for the LBG clustering algorithm. If true, the global optimization is always run after a single cluster has been split. If false, several clusters are split within the same step before applying the global optimization. Applying the global optimization less often is faster, but can lead to less optimal results, especially having 2 nearby clusters that could be represented by 1) *)
		hrPrev	:	HRESULT;	(* HRESULT indicating the result of previous operations (If SUCCEEDED(hrPrev) equals false, no operation is executed.) *)
	END_VAR

END_FUNCTION

// Functions/Image Color and Contrast Processing/F_VN_WhiteBalance

	{attribute 'TcIecLibraryType'}
	{attribute 'external_name' := 'F_VN_WhiteBalance_GUID_AFB27543_236C_4A4D_FF99_14E6BF4A61E4'}
	(* Calculates the white balance ratios for a RGB image. Uses the green channel as a reference and computes the relative ratios for the red and blue channels. Requires a non-reflecting, not overexposed white colored object (e.g. a sheet of paper) in at least 100 pixels of the image to provide reasonable results. The resulting ratios can then be set on the camera (multiply with existing ratios), or applied in the PLC via MultiplyImageWithVector. *)
	FUNCTION F_VN_WhiteBalance : HRESULT
	VAR_INPUT
		ipSrcImage	:	ITcVnImage;	(* Source image (3 channels (RGB), USINT or UINT) *)
		ipDestImage	:	REFERENCE TO ITcVnImage;	(* Destination image with white balance applied (optional, set to 0 if not required. An appropriate image will be created if required.) *)
		fRatioRed	:	REFERENCE TO REAL;	(* Returns the ratio for the red channel *)
		fRatioBlue	:	REFERENCE TO REAL;	(* Returns the ratio for the blue channel *)
		nMaxValue	:	UDINT;	(* Specify the maximum pixel value that would be achieved by overexposure (usually 255 for 8 bit or 4095 for 12 bit data) *)
		hrPrev	:	HRESULT;	(* HRESULT indicating the result of previous operations (If SUCCEEDED(hrPrev) equals false, no operation is executed.) *)
	END_VAR

END_FUNCTION

// Functions/Contour Analysis/F_VN_ApproximatePolygon

	{attribute 'TcIecLibraryType'}
	{attribute 'external_name' := 'F_VN_ApproximatePolygon_GUID_93C71A1C_1EC2_47AB_D7BC_225D41873114'}
	(* Approximate a contour to a simplified polygon (using the Douglas-Peucker algorithm). *)
	FUNCTION F_VN_ApproximatePolygon : HRESULT
	VAR_INPUT
		ipSrcContour	:	ITcVnContainer;	(* Single contour (ContainerType_Vector_TcVnPoint2_DINT or ContainerType_Vector_TcVnPoint2_REAL; The elements of this container are the points of the contour.) *)
		ipDestContour	:	REFERENCE TO ITcVnContainer;	(* Returns a container which is filled with the approximated polygon points (same type ID as ipSrcContour; Non-zero interface pointers are reused.) *)
		fMaxDist	:	LREAL;	(* Maximum distance between the original contour and its approximation *)
		bClosed	:	BOOL;	(* Specify, if the contour is closed (first and last points connected) or not *)
		hrPrev	:	HRESULT;	(* HRESULT indicating the result of previous operations (If SUCCEEDED(hrPrev) equals false, no operation is executed.) *)
	END_VAR

END_FUNCTION

// Functions/Contour Analysis/F_VN_CheckIfPointIsInsideContour

	{attribute 'TcIecLibraryType'}
	{attribute 'external_name' := 'F_VN_CheckIfPointIsInsideContour_GUID_56C21A47_19B7_49C0_CBA1_CEB6C1D33BA6'}
	(* Checks if a point is inside a contour (and optionally return the distance to it). *)
	FUNCTION F_VN_CheckIfPointIsInsideContour : HRESULT
	VAR_INPUT
		ipContour	:	ITcVnContainer;	(* Single contour (ContainerType_Vector_TcVnPoint2_DINT or ContainerType_Vector_TcVnPoint2_REAL) *)
	END_VAR
	VAR_IN_OUT
		aPoint	:	TcVnPoint2_REAL;	(* Point position to check *)
		fDist	:	LREAL;	(* Returns the result (> 0: the point is inside the contour; 0: the point is on the contour; < 0: the point is outside the contour) *)
	END_VAR
	VAR_INPUT
		bMeasureDistance	:	BOOL;	(* If true, fDist returns the distance to the nearest contour edge. Otherwise, fDist only returns -1, 0 or +1 (recommended to set to false if the distance is not required, as this is faster). *)
		hrPrev	:	HRESULT;	(* HRESULT indicating the result of previous operations (If SUCCEEDED(hrPrev) equals false, no operation is executed.) *)
	END_VAR

END_FUNCTION

// Functions/Contour Analysis/F_VN_ContourArea

	{attribute 'TcIecLibraryType'}
	{attribute 'external_name' := 'F_VN_ContourArea_GUID_8708408E_9C3A_40CE_E164_942A10918438'}
	(* Estimate the contour area using Green's formula. *)
	FUNCTION F_VN_ContourArea : HRESULT
	VAR_INPUT
		ipContour	:	ITcVnContainer;	(* Single contour (ContainerType_Vector_TcVnPoint2_DINT or ContainerType_Vector_TcVnPoint2_REAL; The elements of this container are the points of the contour.) *)
	END_VAR
	VAR_IN_OUT
		fArea	:	LREAL;	(* Returns the estimated contour area (The actual contour area may differ depending on the shape of the contour.) *)
	END_VAR
	VAR_INPUT
		hrPrev	:	HRESULT;	(* HRESULT indicating the result of previous operations (If SUCCEEDED(hrPrev) equals false, no operation is executed.) *)
	END_VAR

END_FUNCTION

// Functions/Contour Analysis/F_VN_ContourCenterOfMass

	{attribute 'TcIecLibraryType'}
	{attribute 'external_name' := 'F_VN_ContourCenterOfMass_GUID_3B6C1ADF_386F_4431_F62D_62C98D51C305'}
	(* Computes the center of mass of a contour. *)
	FUNCTION F_VN_ContourCenterOfMass : HRESULT
	VAR_INPUT
		ipContour	:	ITcVnContainer;	(* Single contour (ContainerType_Vector_TcVnPoint2_DINT or ContainerType_Vector_TcVnPoint2_REAL; The elements of this container are the points of the contour.) *)
	END_VAR
	VAR_IN_OUT
		aCenterOfMass	:	TcVnPoint2_LREAL;	(* Returns the center of mass of the contour *)
	END_VAR
	VAR_INPUT
		hrPrev	:	HRESULT;	(* HRESULT indicating the result of previous operations (If SUCCEEDED(hrPrev) equals false, no operation is executed.) *)
	END_VAR

END_FUNCTION

// Functions/Contour Analysis/F_VN_ContourCircularity

	{attribute 'TcIecLibraryType'}
	{attribute 'external_name' := 'F_VN_ContourCircularity_GUID_C187ACD8_3DE8_4CFB_F8F5_6189C13AA123'}
	(* Computes the circularity of a contour (1.0: ideal circle, 0.0: straight line). *)
	FUNCTION F_VN_ContourCircularity : HRESULT
	VAR_INPUT
		ipContour	:	ITcVnContainer;	(* Single contour (ContainerType_Vector_TcVnPoint2_DINT or ContainerType_Vector_TcVnPoint2_REAL; The elements of this container are the points of the contour.) *)
	END_VAR
	VAR_IN_OUT
		fCircularity	:	LREAL;	(* Returns the circularity of the contour [0..1] *)
	END_VAR
	VAR_INPUT
		hrPrev	:	HRESULT;	(* HRESULT indicating the result of previous operations (If SUCCEEDED(hrPrev) equals false, no operation is executed.) *)
	END_VAR

END_FUNCTION

// Functions/Contour Analysis/F_VN_ContourConvexity

	{attribute 'TcIecLibraryType'}
	{attribute 'external_name' := 'F_VN_ContourConvexity_GUID_2FE93699_1A61_4B78_DE53_67FEE13C2168'}
	(* Computes the convexity of a contour as the ratio between the contour's area and the area of the convex hull (1.0: convex shapes (i.e. rectangle, circle, ..., etc.), 0.0: zero area (i.e. a line or an empty contour)). *)
	FUNCTION F_VN_ContourConvexity : HRESULT
	VAR_INPUT
		ipContour	:	ITcVnContainer;	(* Single contour (ContainerType_Vector_TcVnPoint2_DINT or ContainerType_Vector_TcVnPoint2_REAL; The elements of this container are the points of the contour.) *)
	END_VAR
	VAR_IN_OUT
		fConvexity	:	LREAL;	(* Returns the convexity of the contour [0..1] *)
	END_VAR
	VAR_INPUT
		hrPrev	:	HRESULT;	(* HRESULT indicating the result of previous operations (If SUCCEEDED(hrPrev) equals false, no operation is executed.) *)
	END_VAR

END_FUNCTION

// Functions/Contour Analysis/F_VN_ContourEccentricity

	{attribute 'TcIecLibraryType'}
	{attribute 'external_name' := 'F_VN_ContourEccentricity_GUID_A0353137_C866_45BA_D4D9_C86D13C064E9'}
	(* Computes the eccentricity of a contour (0.0: circular, 1.0: linear). *)
	FUNCTION F_VN_ContourEccentricity : HRESULT
	VAR_INPUT
		ipContour	:	ITcVnContainer;	(* Single contour (ContainerType_Vector_TcVnPoint2_DINT or ContainerType_Vector_TcVnPoint2_REAL; The elements of this container are the points of the contour.) *)
	END_VAR
	VAR_IN_OUT
		fEccentricity	:	LREAL;	(* Returns the eccentricity of the contour [0..1] *)
	END_VAR
	VAR_INPUT
		hrPrev	:	HRESULT;	(* HRESULT indicating the result of previous operations (If SUCCEEDED(hrPrev) equals false, no operation is executed.) *)
	END_VAR

END_FUNCTION

// Functions/Contour Analysis/F_VN_ContourElongation

	{attribute 'TcIecLibraryType'}
	{attribute 'external_name' := 'F_VN_ContourElongation_GUID_0D32A294_1416_4359_D2C2_FFE6EE05D015'}
	(* Computes the elongation factor of a contour. *)
	FUNCTION F_VN_ContourElongation : HRESULT
	VAR_INPUT
		ipContour	:	ITcVnContainer;	(* Single contour (ContainerType_Vector_TcVnPoint2_DINT or ContainerType_Vector_TcVnPoint2_REAL; The elements of this container are the points of the contour.) *)
	END_VAR
	VAR_IN_OUT
		fElongation	:	LREAL;	(* Returns the elongation of the contour *)
	END_VAR
	VAR_INPUT
		hrPrev	:	HRESULT;	(* HRESULT indicating the result of previous operations (If SUCCEEDED(hrPrev) equals false, no operation is executed.) *)
	END_VAR

END_FUNCTION

// Functions/Contour Analysis/F_VN_ContourExtremePoint

	{attribute 'TcIecLibraryType'}
	{attribute 'external_name' := 'F_VN_ContourExtremePoint_GUID_D09123FB_2E1E_4AFD_D9E8_D30E1F6E76C2'}
	(* Finds the contour extreme point. *)
	FUNCTION F_VN_ContourExtremePoint : HRESULT
	VAR_INPUT
		ipContour	:	ITcVnContainer;	(* Source container with 2D points (TcVnPoint2_DINT or TcVnPoint2_REAL or TcVnPoint2_LREAL) *)
		eDirection	:	ETcVnExtremePointDirection;	(* Selects the search direction for the extreme point *)
	END_VAR
	VAR_IN_OUT
		aExtremePoint	:	TcVnPoint2_LREAL;	(* Returns the extreme point of the contour, according to eDirection *)
	END_VAR
	VAR_INPUT
		hrPrev	:	HRESULT;	(* HRESULT indicating the result of previous operations (If SUCCEEDED(hrPrev) equals false, no operation is executed.) *)
	END_VAR

END_FUNCTION

// Functions/Contour Analysis/F_VN_ContourInertiaRatio

	{attribute 'TcIecLibraryType'}
	{attribute 'external_name' := 'F_VN_ContourInertiaRatio_GUID_C82A5936_228A_4565_C34D_8F7AF49D8D2A'}
	(* Computes the inertia ratio of a contour which reflects how a contour/shape is elongated (i.e. circle: 1.0, line: 0.0). *)
	FUNCTION F_VN_ContourInertiaRatio : HRESULT
	VAR_INPUT
		ipContour	:	ITcVnContainer;	(* Single contour (ContainerType_Vector_TcVnPoint2_DINT or ContainerType_Vector_TcVnPoint2_REAL; The elements of this container are the points of the contour.) *)
	END_VAR
	VAR_IN_OUT
		fInertiaRatio	:	LREAL;	(* Returns the inertia raio of the contour [0..1] *)
	END_VAR
	VAR_INPUT
		hrPrev	:	HRESULT;	(* HRESULT indicating the result of previous operations (If SUCCEEDED(hrPrev) equals false, no operation is executed.) *)
	END_VAR

END_FUNCTION

// Functions/Contour Analysis/F_VN_ContourMoments

	{attribute 'TcIecLibraryType'}
	{attribute 'external_name' := 'F_VN_ContourMoments_GUID_A52ED52C_148B_4D1E_D5CC_CF0DDCCA9AE5'}
	(* Computes the spatial moments, the central moments, and the central normalized moments of a contour up to the third order. *)
	FUNCTION F_VN_ContourMoments : HRESULT
	VAR_INPUT
		ipContour	:	ITcVnContainer;	(* Single contour (ContainerType_Vector_TcVnPoint2_DINT or ContainerType_Vector_TcVnPoint2_REAL; The elements of this container are the points of the contour.) *)
	END_VAR
	VAR_IN_OUT
		stMoments	:	TcVnMoments;	(* Returns a struct containing the moments *)
	END_VAR
	VAR_INPUT
		hrPrev	:	HRESULT;	(* HRESULT indicating the result of previous operations (If SUCCEEDED(hrPrev) equals false, no operation is executed.) *)
	END_VAR

END_FUNCTION

// Functions/Contour Analysis/F_VN_ContourOrientation

	{attribute 'TcIecLibraryType'}
	{attribute 'external_name' := 'F_VN_ContourOrientation_GUID_D129B24C_7E46_4F7E_E2E3_8AE97B2ABE95'}
	(* Calculate the orientation of a contour or a set of points. *)
	FUNCTION F_VN_ContourOrientation : HRESULT
	VAR_INPUT
		ipContour	:	ITcVnContainer;	(* Source point set (ContainerType_Vector_TcVnPoint2_DINT, ContainerType_Vector_TcVnPoint2_REAL, or ContainerType_Vector_TcVnPoint2_LREAL. The elements of this container are the individual points.) *)
	END_VAR
	VAR_IN_OUT
		stOrientation	:	TcVnRotatedRectangle;	(* Resulting rotated rectangle, containig center of mass, lenghts of axes, and rotation angle of the contour in clockwise direction. *)
	END_VAR
	VAR_INPUT
		hrPrev	:	HRESULT;	(* HRESULT indicating the result of previous operations (If SUCCEEDED(hrPrev) equals false, no operation is executed.) *)
	END_VAR

END_FUNCTION

// Functions/Contour Analysis/F_VN_ContourOrientationExp

	{attribute 'TcIecLibraryType'}
	{attribute 'external_name' := 'F_VN_ContourOrientationExp_GUID_05090D1D_BEF9_4DEE_CC7C_74C9969B8B2D'}
	(* Calculate the orientation of a contour or a set of points. (expert function) *)
	FUNCTION F_VN_ContourOrientationExp : HRESULT
	VAR_INPUT
		ipContour	:	ITcVnContainer;	(* Source point set (ContainerType_Vector_TcVnPoint2_DINT, ContainerType_Vector_TcVnPoint2_REAL, or ContainerType_Vector_TcVnPoint2_LREAL. The elements of this container are the individual points.) *)
	END_VAR
	VAR_IN_OUT
		stOrientation	:	TcVnRotatedRectangle;	(* Resulting rotated rectangle, containig center of mass, lenghts of axes, and rotation angle of the contour in clockwise direction. *)
	END_VAR
	VAR_INPUT
		eMethod	:	ETcVnOrientationMethod;	(* Method for calculating the orientation.  *)
		hrPrev	:	HRESULT;	(* HRESULT indicating the result of previous operations (If SUCCEEDED(hrPrev) equals false, no operation is executed.) *)
	END_VAR

END_FUNCTION

// Functions/Contour Analysis/F_VN_ContourPerimeter

	{attribute 'TcIecLibraryType'}
	{attribute 'external_name' := 'F_VN_ContourPerimeter_GUID_95B5DD79_9C08_49D3_D12B_0E74B7283D82'}
	(* Computes the perimeter of a contour (curve length if the contour is not closed). *)
	FUNCTION F_VN_ContourPerimeter : HRESULT
	VAR_INPUT
		ipContour	:	ITcVnContainer;	(* Single contour (ContainerType_Vector_TcVnPoint2_DINT or ContainerType_Vector_TcVnPoint2_REAL; The elements of this container are the points of the contour.) *)
	END_VAR
	VAR_IN_OUT
		fPerimeter	:	LREAL;	(* Returns the perimeter of the contour *)
	END_VAR
	VAR_INPUT
		bClosed	:	BOOL;	(* Specifys, if the contour is closed (first and last points connected) or not *)
		hrPrev	:	HRESULT;	(* HRESULT indicating the result of previous operations (If SUCCEEDED(hrPrev) equals false, no operation is executed.) *)
	END_VAR

END_FUNCTION

// Functions/Contour Analysis/F_VN_ContourRoundness

	{attribute 'TcIecLibraryType'}
	{attribute 'external_name' := 'F_VN_ContourRoundness_GUID_56C6EC9D_0E5F_406B_CF02_87F34B0AB5F5'}
	(* Computes the roundness of a contour (perimeter^2 / area). *)
	FUNCTION F_VN_ContourRoundness : HRESULT
	VAR_INPUT
		ipContour	:	ITcVnContainer;	(* Single contour (ContainerType_Vector_TcVnPoint2_DINT or ContainerType_Vector_TcVnPoint2_REAL; The elements of this container are the points of the contour.) *)
	END_VAR
	VAR_IN_OUT
		fRoundness	:	LREAL;	(* Returns the roundness of the contour *)
	END_VAR
	VAR_INPUT
		hrPrev	:	HRESULT;	(* HRESULT indicating the result of previous operations (If SUCCEEDED(hrPrev) equals false, no operation is executed.) *)
	END_VAR

END_FUNCTION

// Functions/Contour Analysis/F_VN_ConvexHullPoints

	{attribute 'TcIecLibraryType'}
	{attribute 'external_name' := 'F_VN_ConvexHullPoints_GUID_0C61FAB4_B908_4095_D5BE_039E6E82BCE1'}
	(* Determines the convex hull of a point set. *)
	FUNCTION F_VN_ConvexHullPoints : HRESULT
	VAR_INPUT
		ipPointSet	:	ITcVnContainer;	(* Source point set (ContainerType_Vector_TcVnPoint2_DINT or ContainerType_Vector_TcVnPoint2_REAL; The elements of this container are the individual points.) *)
		ipConvexHull	:	REFERENCE TO ITcVnContainer;	(* Returns a container which is filled with the sorted convex hull points (same type ID as ipPointSet; Non-zero interface pointers are reused.) *)
		hrPrev	:	HRESULT;	(* HRESULT indicating the result of previous operations (If SUCCEEDED(hrPrev) equals false, no operation is executed.) *)
	END_VAR

END_FUNCTION

// Functions/Contour Analysis/F_VN_ConvexHullPointsExp

	{attribute 'TcIecLibraryType'}
	{attribute 'external_name' := 'F_VN_ConvexHullPointsExp_GUID_41D1F5D6_E57E_47C0_EA24_8690B8D47508'}
	(* Determines the convex hull of a point set. (expert function) *)
	FUNCTION F_VN_ConvexHullPointsExp : HRESULT
	VAR_INPUT
		ipPointSet	:	ITcVnContainer;	(* Source point set (ContainerType_Vector_TcVnPoint2_DINT or ContainerType_Vector_TcVnPoint2_REAL; The elements of this container are the individual points.) *)
		ipConvexHull	:	REFERENCE TO ITcVnContainer;	(* Returns a container which is filled with the sorted convex hull points (same type ID as ipPointSet; Non-zero interface pointers are reused.) *)
		bClockwise	:	BOOL;	(* Selects the sorting direction of the hull points, assuming cartesian coordinates. *)
		hrPrev	:	HRESULT;	(* HRESULT indicating the result of previous operations (If SUCCEEDED(hrPrev) equals false, no operation is executed.) *)
	END_VAR

END_FUNCTION

// Functions/Contour Analysis/F_VN_ConvexityDefects

	{attribute 'TcIecLibraryType'}
	{attribute 'external_name' := 'F_VN_ConvexityDefects_GUID_8B73B366_0E88_4680_DE70_C94CE8E47F6B'}
	(* Finds the convexity defects of a point set. *)
	FUNCTION F_VN_ConvexityDefects : HRESULT
	VAR_INPUT
		ipContour	:	ITcVnContainer;	(* Source contour (ContainerType_Vector_TcVnPoint2_DINT; The elements of this container are the individual points.) *)
		ipConvexityDefects	:	REFERENCE TO ITcVnContainer;	(* Returns a container which is filled with the convexity defects (ContainerType_Vector_TcVnVector4_DINT with [startIndex, endIndex, furthestPointIndex, fixedPointDistance (8 fraction bits, i.e. divide by 256 to get the distance in pixels)]; Non-zero interface pointers are reused.) *)
		hrPrev	:	HRESULT;	(* HRESULT indicating the result of previous operations (If SUCCEEDED(hrPrev) equals false, no operation is executed.) *)
	END_VAR

END_FUNCTION

// Functions/Contour Analysis/F_VN_CustomElementWiseContainerOperation_ITcVnContainer

	{attribute 'TcIecLibraryType'}
	{attribute 'external_name' := 'F_VN_CustomElementWiseContainerOperation_ITcVnContainer_GUID_D4B8C76E_3323_48F3_E04E_DCCB0A26F4C8'}
	(* Performs a custom, element wise operation on a set of up to 3 containers. *)
	FUNCTION F_VN_CustomElementWiseContainerOperation_ITcVnContainer : HRESULT
	VAR_INPUT
		ipContainer1	:	ITcVnContainer;	(* Container 1 *)
		ipContainer2	:	ITcVnContainer;	(* Container 2 *)
		ipContainer3	:	ITcVnContainer;	(* Container 3 *)
		ipOperationFB	:	ITcVnCustomContainerOperation_ITcVnContainer;	(* Custom operation on the container elements *)
		hrPrev	:	HRESULT;	(* HRESULT indicating the result of previous operations (If SUCCEEDED(hrPrev) equals false, no operation is executed.) *)
	END_VAR

END_FUNCTION

// Interfaces/Containers/Function Blocks/ITcVnCustomContainerOperation_ITcVnContainer

	(* Offers an interface for custom, elementwise container operations (for containers of containers) with up to 3 different containers. *)
	{attribute 'c++_compatible'}
	INTERFACE ITcVnCustomContainerOperation_ITcVnContainer


(* Executes the custom operation on the container elements. *)
	{attribute 'c++_compatible'}
	{attribute 'minimal_input_size' := '4'}
	{attribute 'pack_mode' := '4'}
	METHOD Execute : HRESULT
	VAR_INPUT
		ipElement1 : ITcVnContainer;
		ipElement2 : ITcVnContainer;
		ipElement3 : ITcVnContainer;
	END_VAR
END_METHOD

END_INTERFACE

// Functions/Contour Analysis/F_VN_CustomElementWiseContainerOperation_ITcVnForwardIterator

	{attribute 'TcIecLibraryType'}
	{attribute 'external_name' := 'F_VN_CustomElementWiseContainerOperation_ITcVnForwardIterator_GUID_FC12F199_52D7_48F7_F7BB_FC8DF6704071'}
	(* Performs a custom, element wise operation on a set of up to 3 containers. *)
	FUNCTION F_VN_CustomElementWiseContainerOperation_ITcVnForwardIterator : HRESULT
	VAR_INPUT
		ipContainer1	:	ITcVnContainer;	(* Container 1 *)
		ipContainer2	:	ITcVnContainer;	(* Container 2 *)
		ipContainer3	:	ITcVnContainer;	(* Container 3 *)
		ipOperationFB	:	ITcVnCustomContainerOperation_ITcVnForwardIterator;	(* Custom operation on the elements *)
		hrPrev	:	HRESULT;	(* HRESULT indicating the result of previous operations (If SUCCEEDED(hrPrev) equals false, no operation is executed.) *)
	END_VAR

END_FUNCTION

// Interfaces/Containers/Function Blocks/ITcVnCustomContainerOperation_ITcVnForwardIterator

	(* Offers an interface for custom, elementwise container operations with up to 3 different containers. *)
	{attribute 'c++_compatible'}
	INTERFACE ITcVnCustomContainerOperation_ITcVnForwardIterator


(* Executes the custom operation on the container elements. *)
	{attribute 'c++_compatible'}
	{attribute 'minimal_input_size' := '4'}
	{attribute 'pack_mode' := '4'}
	METHOD Execute : HRESULT
	VAR_INPUT
		ipElement1 : ITcVnForwardIterator;
		ipElement2 : ITcVnForwardIterator;
		ipElement3 : ITcVnForwardIterator;
	END_VAR
END_METHOD

END_INTERFACE

// Functions/Contour Analysis/F_VN_EnclosingCircle

	{attribute 'TcIecLibraryType'}
	{attribute 'external_name' := 'F_VN_EnclosingCircle_GUID_73AEFE24_1294_4160_E1B9_CEBEA99C97A4'}
	(* Searchs for a minimum area circle enclosing a set of points. *)
	FUNCTION F_VN_EnclosingCircle : HRESULT
	VAR_INPUT
		ipPointSet	:	ITcVnContainer;	(* Source point set (ContainerType_Vector_TcVnPoint2_DINT or ContainerType_Vector_TcVnPoint2_REAL; The elements of this container are the individual points.) *)
	END_VAR
	VAR_IN_OUT
		aCenter	:	TcVnPoint2_REAL;	(* Returns the center of the circle *)
		fRadius	:	REAL;	(* Returns the radius of the circle *)
	END_VAR
	VAR_INPUT
		hrPrev	:	HRESULT;	(* HRESULT indicating the result of previous operations (If SUCCEEDED(hrPrev) equals false, no operation is executed.) *)
	END_VAR

END_FUNCTION

// Functions/Contour Analysis/F_VN_EnclosingRectangle

	{attribute 'TcIecLibraryType'}
	{attribute 'external_name' := 'F_VN_EnclosingRectangle_GUID_05F99E57_B583_450F_F9FF_EF4C035C9024'}
	(* Searches for a minimum area rectangle enclosing a set of points. *)
	FUNCTION F_VN_EnclosingRectangle : HRESULT
	VAR_INPUT
		ipPointSet	:	ITcVnContainer;	(* Source point set (ContainerType_Vector_TcVnPoint2_DINT or ContainerType_Vector_TcVnPoint2_REAL; The elements of this container are the individual points.) *)
	END_VAR
	VAR_IN_OUT
		stRectangle	:	TcVnRotatedRectangle;	(* Returns the determined rectangle *)
	END_VAR
	VAR_INPUT
		hrPrev	:	HRESULT;	(* HRESULT indicating the result of previous operations (If SUCCEEDED(hrPrev) equals false, no operation is executed.) *)
	END_VAR

END_FUNCTION

// Functions/Contour Analysis/F_VN_EnclosingTriangle

	{attribute 'TcIecLibraryType'}
	{attribute 'external_name' := 'F_VN_EnclosingTriangle_GUID_C8053409_6969_4B70_DC50_8DC5F1F409DE'}
	(* Searches for a minimum area triangle enclosing a set of points. *)
	FUNCTION F_VN_EnclosingTriangle : HRESULT
	VAR_INPUT
		ipPointSet	:	ITcVnContainer;	(* Source point set (ContainerType_Vector_TcVnPoint2_DINT or ContainerType_Vector_TcVnPoint2_REAL; The elements of this container are the individual points.) *)
	END_VAR
	VAR_IN_OUT
		aTriangleVertices	:	TcVnArray3_Point2_REAL;	(* Returns the 3 triangle vertices *)
	END_VAR
	VAR_INPUT
		hrPrev	:	HRESULT;	(* HRESULT indicating the result of previous operations (If SUCCEEDED(hrPrev) equals false, no operation is executed.) *)
	END_VAR
	VAR_OUTPUT
		fArea	:	LREAL;	(* Returns the triangle area *)
	END_VAR

END_FUNCTION

// Functions/Contour Analysis/F_VN_FitEllipse

	{attribute 'TcIecLibraryType'}
	{attribute 'external_name' := 'F_VN_FitEllipse_GUID_CEB11D46_E443_41D2_E0CD_64439F69F990'}
	(* Fit an ellipse in a point set. *)
	FUNCTION F_VN_FitEllipse : HRESULT
	VAR_INPUT
		ipPointSet	:	ITcVnContainer;	(* Source point set (ContainerType_Vector_TcVnPoint2_DINT or ContainerType_Vector_TcVnPoint2_REAL; At least 5 reasonable points are required! The elements of this container are the individual points.) *)
	END_VAR
	VAR_IN_OUT
		stEllipse	:	TcVnRotatedRectangle;	(* Resulting ellipse, described by a rotated rectangle. *)
	END_VAR
	VAR_INPUT
		hrPrev	:	HRESULT;	(* HRESULT indicating the result of previous operations (If SUCCEEDED(hrPrev) equals false, no operation is executed.) *)
	END_VAR

END_FUNCTION

// Functions/Contour Analysis/F_VN_FitLine

	{attribute 'TcIecLibraryType'}
	{attribute 'external_name' := 'F_VN_FitLine_GUID_EEA7AB17_D765_4AE5_C52B_3F172D4F5835'}
	(* Fit a line into a point set. *)
	FUNCTION F_VN_FitLine : HRESULT
	VAR_INPUT
		ipPointSet	:	ITcVnContainer;	(* Source point set (ContainerType_Vector_TcVnPoint2_DINT or ContainerType_Vector_TcVnPoint2_REAL; The elements of this container are the individual points.) *)
	END_VAR
	VAR_IN_OUT
		aFitLine	:	TcVnVector4_LREAL;	(* Resulting line. The first and second element describe the x and y component of a vector collinear to the line. The third and fourth element describe the x and y component of a point on the line. *)
	END_VAR
	VAR_INPUT
		hrPrev	:	HRESULT;	(* HRESULT indicating the result of previous operations (If SUCCEEDED(hrPrev) equals false, no operation is executed.) *)
	END_VAR

END_FUNCTION

// Functions/Contour Analysis/F_VN_FitLineExp

	{attribute 'TcIecLibraryType'}
	{attribute 'external_name' := 'F_VN_FitLineExp_GUID_266CAEED_F24E_4142_FD97_F103F8A2EE41'}
	(* Fit a line into a point set. (expert function) *)
	FUNCTION F_VN_FitLineExp : HRESULT
	VAR_INPUT
		ipPointSet	:	ITcVnContainer;	(* Source point set (ContainerType_Vector_TcVnPoint2_DINT or ContainerType_Vector_TcVnPoint2_REAL; The elements of this container are the individual points.) *)
	END_VAR
	VAR_IN_OUT
		aFitLine	:	TcVnVector4_LREAL;	(* Resulting line. The first and second element describe the x and y component of a vector collinear to the line. The third and fourth element describe the x and y component of a point on the line. *)
	END_VAR
	VAR_INPUT
		eDistanceType	:	ETcVnDistanceType;	(* Distance computation method (supported: L1, L2, L12, FAIR, WELSCH, HUBER) *)
		fParam	:	LREAL;	(* Numerical parameter (c) for some eDistanceType (should be >= 0). If 0, an optimal value is chosen internally. *)
		fEpsRadius	:	LREAL;	(* Accuracy of the radius (distance of the line from the coordinate origin, should be > 0). A smaller value means higher accuracy. *)
		fEpsAngle	:	LREAL;	(* Accuracy of the angle (should be > 0). A smaller value means higher accuracy. *)
		hrPrev	:	HRESULT;	(* HRESULT indicating the result of previous operations (If SUCCEEDED(hrPrev) equals false, no operation is executed.) *)
	END_VAR

END_FUNCTION

// Functions/Contour Analysis/F_VN_FourierDescriptors

	{attribute 'TcIecLibraryType'}
	{attribute 'external_name' := 'F_VN_FourierDescriptors_GUID_77D62952_5594_4CAC_D61A_056B6D5BCFBD'}
	(* Computes the fourier descriptors for a closed contour. *)
	FUNCTION F_VN_FourierDescriptors : HRESULT
	VAR_INPUT
		ipContour	:	ITcVnContainer;	(* Closed contour (ContainerType_Vector_TcVnPoint2_DINT or ContainerType_Vector_TcVnPoint2_REAL or ContainerType_Vector_TcVnPoint2_LREAL. Providing the full contour is strongly recommended, i.e. use TCVN_CAM_NONE for contour detection algorithms.) *)
		ipDescriptors	:	REFERENCE TO ITcVnContainer;	(* Returns the fourier descriptors for ipContour (Re0, Im0, Re1, Im1, ...; ContainerType_Vector_LREAL if ipContour is of type ContainerType_Vector_TcVnPoint2_LREAL, else ContainerType_Vector_REAL.) *)
		nDescriptors	:	DINT;	(* Specifies how many descriptors should be returned (set to -1 to return all computed descriptors, i.e. at least as many as the number of contour points) *)
		hrPrev	:	HRESULT;	(* HRESULT indicating the result of previous operations (If SUCCEEDED(hrPrev) equals false, no operation is executed.) *)
	END_VAR

END_FUNCTION

// Functions/Contour Analysis/F_VN_MatchContours

	{attribute 'TcIecLibraryType'}
	{attribute 'external_name' := 'F_VN_MatchContours_GUID_985D7BEE_9272_4D8E_D362_C6613FD43A18'}
	(* Compare contours using the Hu moment invariants. In case of multiple contours in each container, the best matches are found and the average dissimilarity over all matched contours is returned. *)
	FUNCTION F_VN_MatchContours : HRESULT
	VAR_INPUT
		ipContour1	:	ITcVnContainer;	(* First contour (ContainerType_Vector_TcVnPoint2_DINT or ContainerType_Vector_TcVnPoint2_REAL; The elements of this container are the points of the contour) or collection of multiple contours (ContainerType_Vector_Vector_TcVnPoint2_DINT) *)
		ipContour2	:	ITcVnContainer;	(* Second contour (same type as ipContour1) *)
		eComparisonMethod	:	ETcVnContoursMatchComparisonMethod;	(* Method used for comparing the Hu moment invariants of the contours *)
	END_VAR
	VAR_IN_OUT
		fDissimilarity	:	LREAL;	(* Returns the dissimilarity of the contours depending on the chosen comparison method *)
	END_VAR
	VAR_INPUT
		hrPrev	:	HRESULT;	(* HRESULT indicating the result of previous operations (If SUCCEEDED(hrPrev) equals false, no operation is executed.) *)
	END_VAR

END_FUNCTION

// Functions/Contour Analysis/F_VN_MatchContoursExp

	{attribute 'TcIecLibraryType'}
	{attribute 'external_name' := 'F_VN_MatchContoursExp_GUID_E926429A_9DFE_4596_D583_A2F41D58F27F'}
	(* Compare contours using the Hu moment invariants (and optionally further aspects). In case of multiple contours in each container, the best matches are found and the average dissimilarity over all matched contours is returned. (expert function) *)
	FUNCTION F_VN_MatchContoursExp : HRESULT
	VAR_INPUT
		ipContour1	:	ITcVnContainer;	(* First contour (ContainerType_Vector_TcVnPoint2_DINT or ContainerType_Vector_TcVnPoint2_REAL; The elements of this container are the points of the contour) or collection of multiple contours (ContainerType_Vector_Vector_TcVnPoint2_DINT) *)
		ipContour2	:	ITcVnContainer;	(* Second contour (same type as ipContour1) *)
		eComparisonMethod	:	ETcVnContoursMatchComparisonMethod;	(* Method used for comparing the Hu moment invariants of the contours *)
	END_VAR
	VAR_IN_OUT
		fDissimilarity	:	LREAL;	(* Returns the dissimilarity of the contours depending on the chosen comparison method *)
	END_VAR
	VAR_INPUT
		fAreaFactor	:	LREAL;	(* If > 0, the relative area difference between contours is scaled by this factor and added to the computed dissimilarity *)
		fAbsPositionFactor	:	LREAL;	(* If > 0, the absolute position difference between contours (i.e. the coordinates of the geometric contour centers) is scaled by this factor and added to the computed dissimilarity *)
		fRelPositionFactor	:	LREAL;	(* If > 0, the relative position difference between contours is scaled by this factor and added to the computed dissimilarity (only used if matching multiple contours) *)
		fNumDiffFactor	:	LREAL;	(* If > 0, the difference between the number of contours in both containers is scaled by this factor and added to the computed dissimilarity (only used if matching multiple contours) *)
		hrPrev	:	HRESULT;	(* HRESULT indicating the result of previous operations (If SUCCEEDED(hrPrev) equals false, no operation is executed.) *)
	END_VAR

END_FUNCTION

// Functions/Contour Analysis/F_VN_MatchContours1vsN

	{attribute 'TcIecLibraryType'}
	{attribute 'external_name' := 'F_VN_MatchContours1vsN_GUID_216BD7F1_E2FD_47A4_E4BA_252424BE5B3D'}
	(* Compare a reference contour with multiple other contours using the Hu moment invariants. Returns a sorted list of best matches. *)
	FUNCTION F_VN_MatchContours1vsN : HRESULT
	VAR_INPUT
		ipRefContour	:	ITcVnContainer;	(* Reference contour (ContainerType_Vector_TcVnPoint2_DINT or ContainerType_Vector_TcVnPoint2_REAL; The elements of this container are the points of the contour) *)
		ipContours	:	ITcVnContainer;	(* Collection of multiple contours (CTcVnContainer_Vector_Vector_TcVnPoint2_DINT) *)
		ipMatchIndexes	:	REFERENCE TO ITcVnContainer;	(* Returns the indexes of the best matches (CTcVnContainer_Vector_ULINT; sorted, first element is best match, i.e. has lowest dissimilarity) *)
		ipDissimilarities	:	REFERENCE TO ITcVnContainer;	(* Returns the computed dissimilarities of the best matches (CTcVnContainer_Vector_LREAL; Optional, set to 0 if not required; sorted corresponding to ipMatchIndexes) *)
		fDissimilarityThreshold	:	LREAL;	(* Neglect irrelevant matches, i.e. dissimilarity > fDissimilarityThreshold *)
		eComparisonMethod	:	ETcVnContoursMatchComparisonMethod;	(* Method used for comparing the Hu moment invariants of the contours *)
		hrPrev	:	HRESULT;	(* HRESULT indicating the result of previous operations (If SUCCEEDED(hrPrev) equals false, no operation is executed.) *)
	END_VAR

END_FUNCTION

// Functions/Contour Analysis/F_VN_MatchContours1vsNExp

	{attribute 'TcIecLibraryType'}
	{attribute 'external_name' := 'F_VN_MatchContours1vsNExp_GUID_6C3FAB14_6CA5_4CAD_D4BD_013EB1315070'}
	(* Compare a reference contour with multiple other contours using the Hu moment invariants (and optionally further aspects). Returns a sorted list of best matches. (expert function) *)
	FUNCTION F_VN_MatchContours1vsNExp : HRESULT
	VAR_INPUT
		ipRefContour	:	ITcVnContainer;	(* Reference contour (ContainerType_Vector_TcVnPoint2_DINT or ContainerType_Vector_TcVnPoint2_REAL; The elements of this container are the points of the contour) *)
		ipContours	:	ITcVnContainer;	(* Collection of multiple contours (CTcVnContainer_Vector_Vector_TcVnPoint2_DINT) *)
		ipMatchIndexes	:	REFERENCE TO ITcVnContainer;	(* Returns the indexes of the best matches (CTcVnContainer_Vector_ULINT; sorted, first element is best match, i.e. has lowest dissimilarity) *)
		ipDissimilarities	:	REFERENCE TO ITcVnContainer;	(* Returns the computed dissimilarities of the best matches (CTcVnContainer_Vector_LREAL; Optional, set to 0 if not required; sorted corresponding to ipMatchIndexes) *)
		fDissimilarityThreshold	:	LREAL;	(* Neglect irrelevant matches, i.e. dissimilarity > fDissimilarityThreshold *)
		eComparisonMethod	:	ETcVnContoursMatchComparisonMethod;	(* Method used for comparing the Hu moment invariants of the contours *)
		fAreaFactor	:	LREAL;	(* If > 0, the relative area difference between contours is scaled by this factor and added to the computed dissimilarity *)
		fAbsPositionFactor	:	LREAL;	(* If > 0, the absolute position difference between contours (i.e. the coordinates of the geometric contour centers) is scaled by this factor and added to the computed dissimilarity *)
		hrPrev	:	HRESULT;	(* HRESULT indicating the result of previous operations (If SUCCEEDED(hrPrev) equals false, no operation is executed.) *)
	END_VAR

END_FUNCTION

// Functions/Contour Analysis/F_VN_UprightBoundingRectangle

	{attribute 'TcIecLibraryType'}
	{attribute 'external_name' := 'F_VN_UprightBoundingRectangle_GUID_2FC75E4C_7ED3_4A18_C935_F5A677F8C0D1'}
	(* Determines the upright bounding rectangle of a set of points. *)
	FUNCTION F_VN_UprightBoundingRectangle : HRESULT
	VAR_INPUT
		ipPointSet	:	ITcVnContainer;	(* Source point set (ContainerType_Vector_TcVnPoint2_DINT or ContainerType_Vector_TcVnPoint2_REAL; The elements of this container are the individual points.) *)
	END_VAR
	VAR_IN_OUT
		stRectangle	:	TcVnRectangle_UDINT;	(* Returns the determined rectangle *)
	END_VAR
	VAR_INPUT
		hrPrev	:	HRESULT;	(* HRESULT indicating the result of previous operations (If SUCCEEDED(hrPrev) equals false, no operation is executed.) *)
	END_VAR

END_FUNCTION

// Functions/Image Filtering/F_VN_BilateralFilter

	{attribute 'TcIecLibraryType'}
	{attribute 'external_name' := 'F_VN_BilateralFilter_GUID_14075620_CBDC_4B35_C56F_18E43E4327CB'}
	(* Apply a Bilateral filter to smooth the image but preserve edges. *)
	FUNCTION F_VN_BilateralFilter : HRESULT
	VAR_INPUT
		ipSrcImage	:	ITcVnImage;	(* Source image *)
		ipDestImage	:	REFERENCE TO ITcVnImage;	(* Destination image (Must be different from ipSrcImage! An appropriate destination image will be created if required.) *)
		nDiameter	:	DINT;	(* Diameter of the pixel neighborhood used for filtering (e.g. 5, 7, 9). If <= 0, it is automatically chosen dependend on fSigmaSpace. *)
		fSigmaColor	:	LREAL;	(* Sigma used for color space filtering (> 0). A larger value means that farther colors are mixed together. *)
		fSigmaSpace	:	LREAL;	(* Sigma used for coordinate space filtering (> 0). A larger value means that farther pixels can influence each other. *)
		hrPrev	:	HRESULT;	(* HRESULT indicating the result of previous operations (If SUCCEEDED(hrPrev) equals false, no operation is executed.) *)
	END_VAR

END_FUNCTION

// Functions/Image Filtering/F_VN_BilateralFilterExp

	{attribute 'TcIecLibraryType'}
	{attribute 'external_name' := 'F_VN_BilateralFilterExp_GUID_E8D103CC_4338_4D9A_FC60_F3148286D208'}
	(* Apply a Bilateral filter to smooth the image but preserve edges. (expert function) *)
	FUNCTION F_VN_BilateralFilterExp : HRESULT
	VAR_INPUT
		ipSrcImage	:	ITcVnImage;	(* Source image *)
		ipDestImage	:	REFERENCE TO ITcVnImage;	(* Destination image (Must be different from ipSrcImage! An appropriate destination image will be created if required.) *)
		nDiameter	:	DINT;	(* Diameter of the pixel neighborhood used for filtering (e.g. 5, 7, 9). If <= 0, it is automatically chosen dependend on fSigmaSpace. *)
		fSigmaColor	:	LREAL;	(* Sigma used for color space filtering (> 0). A larger value means that farther colors are mixed together. *)
		fSigmaSpace	:	LREAL;	(* Sigma used for coordinate space filtering (> 0). A larger value means that farther pixels can influence each other. *)
		eBorderType	:	ETcVnBorderInterpolationMethod;	(* Image border handling *)
		hrPrev	:	HRESULT;	(* HRESULT indicating the result of previous operations (If SUCCEEDED(hrPrev) equals false, no operation is executed.) *)
	END_VAR

END_FUNCTION

// Functions/Image Filtering/F_VN_BoxFilter

	{attribute 'TcIecLibraryType'}
	{attribute 'external_name' := 'F_VN_BoxFilter_GUID_D325D1EC_9D63_40B0_C3EE_07DF9460F83E'}
	(* Apply a box filter to an image. *)
	FUNCTION F_VN_BoxFilter : HRESULT
	VAR_INPUT
		ipSrcImage	:	ITcVnImage;	(* Source image *)
		ipDestImage	:	REFERENCE TO ITcVnImage;	(* Destination image (An appropriate destination image will be created if required.) *)
		nFilterWidth	:	UDINT;	(* Filter width in pixels *)
		nFilterHeight	:	UDINT;	(* Filter height in pixels *)
		hrPrev	:	HRESULT;	(* HRESULT indicating the result of previous operations (If SUCCEEDED(hrPrev) equals false, no operation is executed.) *)
	END_VAR

END_FUNCTION

// Functions/Image Filtering/F_VN_BoxFilterExp

	{attribute 'TcIecLibraryType'}
	{attribute 'external_name' := 'F_VN_BoxFilterExp_GUID_8B873A76_7E14_47C4_E556_B7D7A7C2A503'}
	(* Apply a box filter to an image. (expert function) *)
	FUNCTION F_VN_BoxFilterExp : HRESULT
	VAR_INPUT
		ipSrcImage	:	ITcVnImage;	(* Source image *)
		ipDestImage	:	REFERENCE TO ITcVnImage;	(* Destination image (An appropriate destination image will be created if required.) *)
		nFilterWidth	:	UDINT;	(* Filter width in pixels *)
		nFilterHeight	:	UDINT;	(* Filter height in pixels *)
		eDestDepth	:	ETcVnElementType;	(* Destination image depth *)
	END_VAR
	VAR_IN_OUT
		aAnchor	:	TcVnPoint;	(* Anchor point of the kernel ([-1, -1] for center) *)
	END_VAR
	VAR_INPUT
		bNormalize	:	BOOL;	(* If true, the kernel is normalized by nFilterWidth * nFilterHeight *)
		eBorderType	:	ETcVnBorderInterpolationMethod;	(* Image border handling *)
		hrPrev	:	HRESULT;	(* HRESULT indicating the result of previous operations (If SUCCEEDED(hrPrev) equals false, no operation is executed.) *)
	END_VAR

END_FUNCTION

// Functions/Image Filtering/F_VN_BrightBorderObjects

	{attribute 'TcIecLibraryType'}
	{attribute 'external_name' := 'F_VN_BrightBorderObjects_GUID_F508D8E0_EBBB_4B53_D93F_6DB249AEE805'}
	(* Find bright objects connected to the image border within a gray-scale single-channel image. *)
	FUNCTION F_VN_BrightBorderObjects : HRESULT
	VAR_INPUT
		ipSrcImage	:	ITcVnImage;	(* Source image (USINT, UINT, INT, REAL, or LREAL, 1 channel) *)
		ipDestImage	:	REFERENCE TO ITcVnImage;	(* Destination image (An appropriate destination image will be created if required.) *)
		hrPrev	:	HRESULT;	(* HRESULT indicating the result of previous operations (If SUCCEEDED(hrPrev) equals false, no operation is executed.) *)
	END_VAR

END_FUNCTION

// Functions/Image Filtering/F_VN_CreateStructuringElement

	{attribute 'TcIecLibraryType'}
	{attribute 'external_name' := 'F_VN_CreateStructuringElement_GUID_D7D20D2C_C0FA_409F_E1E0_83EE0E7DDA91'}
	(* Creates a structuring element for the usage with morphological operators and allocate an appropriate data buffer. The initial reference count is set to one if a new image interface is created and kept, otherwise. *)
	FUNCTION F_VN_CreateStructuringElement : HRESULT
	VAR_INPUT
		ipStructuringElement	:	REFERENCE TO ITcVnImage;	(* Returns the created structuring element (Non-zero interface pointers are reused.) *)
		eShape	:	ETcVnStructuringElementShape;	(* Shape of the structuring element (rectangle, cross, or ellipse) *)
		nWidth	:	UDINT;	(* Width *)
		nHeight	:	UDINT;	(* Height *)
		hrPrev	:	HRESULT;	(* HRESULT indicating the result of previous operations (If SUCCEEDED(hrPrev) equals false, no operation is executed.) *)
	END_VAR

END_FUNCTION

// Functions/Image Filtering/F_VN_CustomFilter

	{attribute 'TcIecLibraryType'}
	{attribute 'external_name' := 'F_VN_CustomFilter_GUID_339F1FCF_BE1B_40C4_C211_34A4DA0F0ECE'}
	(* Apply a custom filter to the image. *)
	FUNCTION F_VN_CustomFilter : HRESULT
	VAR_INPUT
		ipSrcImage	:	ITcVnImage;	(* Source image *)
		ipDestImage	:	REFERENCE TO ITcVnImage;	(* Destination image (An appropriate destination image will be created if required.) *)
		eDestDepth	:	ETcVnElementType;	(* Destination image depth *)
	END_VAR
	VAR_IN_OUT
		stKernel	:	TcVnMatrix;	(* Custom filter kernel with values of type REAL or LREAL *)
	END_VAR
	VAR_INPUT
		hrPrev	:	HRESULT;	(* HRESULT indicating the result of previous operations (If SUCCEEDED(hrPrev) equals false, no operation is executed.) *)
	END_VAR

END_FUNCTION

// Functions/Image Filtering/F_VN_CustomFilterExp

	{attribute 'TcIecLibraryType'}
	{attribute 'external_name' := 'F_VN_CustomFilterExp_GUID_1B881621_9971_42A1_F544_8593849F985C'}
	(* Apply a custom filter to the image. (expert function) *)
	FUNCTION F_VN_CustomFilterExp : HRESULT
	VAR_INPUT
		ipSrcImage	:	ITcVnImage;	(* Source image *)
		ipDestImage	:	REFERENCE TO ITcVnImage;	(* Destination image (An appropriate destination image will be created if required.) *)
		eDestDepth	:	ETcVnElementType;	(* Destination image depth *)
	END_VAR
	VAR_IN_OUT
		stKernel	:	TcVnMatrix;	(* Custom filter kernel with values of type REAL or LREAL *)
		aAnchor	:	TcVnPoint;	(* Anchor point of the kernel *)
	END_VAR
	VAR_INPUT
		fDelta	:	LREAL;	(* Value added to each pixel after filtering *)
		eBorderType	:	ETcVnBorderInterpolationMethod;	(* Image border handling *)
		hrPrev	:	HRESULT;	(* HRESULT indicating the result of previous operations (If SUCCEEDED(hrPrev) equals false, no operation is executed.) *)
	END_VAR

END_FUNCTION

// Functions/Image Filtering/F_VN_DarkBorderObjects

	{attribute 'TcIecLibraryType'}
	{attribute 'external_name' := 'F_VN_DarkBorderObjects_GUID_20B4BC89_32B1_4BA8_D571_76C9872FF64B'}
	(* Find dark objects connected to the image border within a gray-scale single-channel image. (equivalent to filling holes) *)
	FUNCTION F_VN_DarkBorderObjects : HRESULT
	VAR_INPUT
		ipSrcImage	:	ITcVnImage;	(* Source image (USINT, UINT, INT, REAL, or LREAL, 1 channel) *)
		ipDestImage	:	REFERENCE TO ITcVnImage;	(* Destination image (An appropriate destination image will be created if required.) *)
		hrPrev	:	HRESULT;	(* HRESULT indicating the result of previous operations (If SUCCEEDED(hrPrev) equals false, no operation is executed.) *)
	END_VAR

END_FUNCTION

